KUKA KRL program: EPS_2_251806_MH47A_A_20260212042244.src

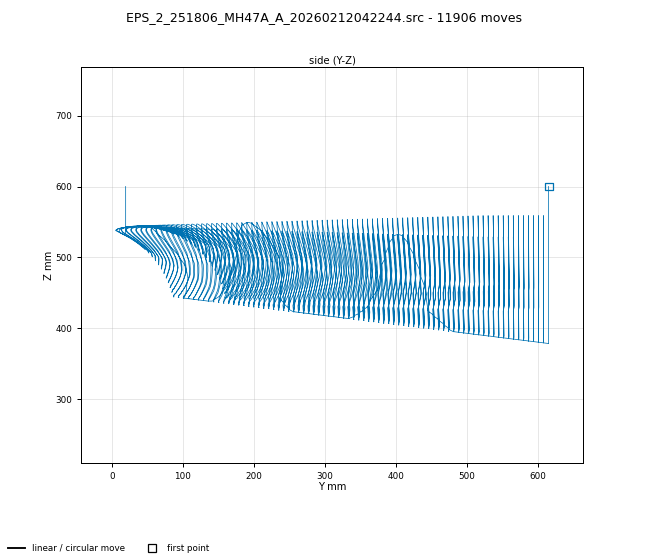
[picture p0: tool path of EPS_2_251806_MH47A_A_20260212042244.src, 11906 of 11908 moves have a stored position in this frame; points joined in program order, loops and branches not executed]
&ACCESS RVP
&REL 4
&COMMENT QRS 19112012
&PARAM EDITMASK = *
DEF PART()
EXT BAS (BAS_COMMAND :IN,REAL :IN )
INT I
BAS (#INITMOV,0 )

;KUKA QRS Post kuka4.cps  Date:22-06-2017 !

File_ID=3019

QRS_PRE_INIT()

;Init var - Until changes are made in qrs_pre_init
Outlet_Square_prg=0
Inlet_1_Square_prg=0
Inlet_2_Square_prg=0
Inlet_3_Square_prg=0
Inlet_4_Square_prg=0
Inlet_5_Square_prg=0

Outlet_1={X 0.000, Y 520.860, Z 458.500, B 0.000, E1 0.000 }
Inlet_1={X 0.000, Y 523.030, Z 428.500, B 0.000, E1 194.000 }
Outlet_1_type=201
Inlet_1_type=201
;QRS#1=Sidecore dimensions
;QRS#2=200-8" PVC SDR 35
;QRS#3=200-8" PVC SDR 35
;QRS#4=
;QRS#5=
;QRS#6=
;QRS#7=
;QRS#8=
;QRS#9=12-08 PSX
;QRS#10=12-08 PSX
;QRS#11=
;QRS#12=
;QRS#13=
;QRS#14=
;QRS#15=
;QRS#16=1220x127x838 2,75'
;QRS#17=EPS Height
;QRS#18=559
;QRS#19=*
;QRS#20= UPDATED VERSION 22-06-2017
;QRS#21=*
Outlet_Square=0100
Inlet_1_Square=0100
Inlet_2_Square=0
Inlet_3_Square=0
Inlet_4_Square=0
Inlet_5_Square=0
Mill_Square=1
Outlet_Square_Prg=204
Inlet_1_Square_prg=204

QRS_INIT()

$ADVANCE=5

; T1
PTP {E1 173.598,E2 173.598}
PTP {X 0,Y 615.497,A -85,B 0,C 180,E1 173.598,E2 173.598,E3 0,E4 0,E5 0,E6 0}
QRS_SPEED_INIT()
LIN {X 0,Y 615.497,Z 600,A -85,B 0,C 180,E1 173.598,E2 173.598,E3 0,E4 0,E5 0,E6 0} C_VEL
LIN {X 0,Y 615.497,Z 388.866,A -85,B 0,C 180,E1 173.598,E2 173.598} C_VEL
LIN {X 0,Y 615.497,Z 380.69,A -85,B 0,C 180,E1 173.598,E2 173.598} C_VEL
LIN {X 0,Y 615.486,Z 378.69,A -85,B 0,C 180,E1 173.412,E2 173.412} C_VEL
LIN {X 0,Y 615.496,Z 378.692,A -85,B 0,C 180,E1 170.801,E2 170.801} C_VEL
LIN {X 0,Y 615.477,Z 378.685,A -85,B 0,C 180,E1 168.139,E2 168.139} C_VEL
LIN {X 0,Y 615.488,Z 378.696,A -85,B 0,C 180,E1 165.451,E2 165.451} C_VEL
LIN {X 0,Y 615.493,Z 378.685,A -85,B 0,C 180,E1 162.73,E2 162.73} C_VEL
LIN {X 0,Y 615.49,Z 378.687,A -85,B 0,C 180,E1 159.967,E2 159.967} C_VEL
LIN {X 0,Y 615.491,Z 378.69,A -85,B 0,C 180,E1 157.156,E2 157.156} C_VEL
LIN {X 0,Y 615.475,Z 378.687,A -85,B 0,C 180,E1 154.431,E2 154.431} C_VEL
LIN {X 0,Y 615.483,Z 378.692,A -85,B 0,C 180,E1 152.085,E2 152.085} C_VEL
LIN {X 0,Y 615.49,Z 378.7,A -85,B 0,C 180,E1 149.84,E2 149.84} C_VEL
LIN {X 0,Y 615.485,Z 378.693,A -85,B 0,C 180,E1 147.542,E2 147.542} C_VEL
LIN {X 0,Y 615.492,Z 378.683,A -85,B 0,C 180,E1 145.185,E2 145.185} C_VEL
LIN {X 0,Y 615.479,Z 378.686,A -85,B 0,C 180,E1 142.757,E2 142.757} C_VEL
LIN {X 0,Y 615.486,Z 378.696,A -85,B 0,C 180,E1 139.91,E2 139.91} C_VEL
LIN {X 0,Y 615.483,Z 378.686,A -85,B 0,C 180,E1 136.952,E2 136.952} C_VEL
LIN {X 0,Y 615.482,Z 378.693,A -85,B 0,C 180,E1 133.997,E2 133.997} C_VEL
LIN {X 0,Y 615.488,Z 378.683,A -85,B 0,C 180,E1 131.473,E2 131.473} C_VEL
LIN {X 0,Y 615.484,Z 378.691,A -85,B 0,C 180,E1 128.903,E2 128.903} C_VEL
LIN {X 0,Y 615.49,Z 378.696,A -85,B 0,C 180,E1 126.424,E2 126.424} C_VEL
LIN {X 0,Y 615.492,Z 378.683,A -85,B 0,C 180,E1 123.535,E2 123.535} C_VEL
LIN {X 0,Y 615.493,Z 378.697,A -85,B 0,C 180,E1 120.919,E2 120.919} C_VEL
LIN {X 0,Y 615.491,Z 378.689,A -85,B 0,C 180,E1 118.451,E2 118.451} C_VEL
LIN {X 0,Y 615.498,Z 378.684,A -85,B 0,C 180,E1 115.571,E2 115.571} C_VEL
LIN {X 0,Y 615.494,Z 378.694,A -85,B 0,C 180,E1 112.844,E2 112.844} C_VEL
LIN {X 0,Y 615.494,Z 378.691,A -85,B 0,C 180,E1 111.431,E2 111.431} C_VEL
LIN {X 0,Y 615.49,Z 382.133,A -85,B 0,C 180,E1 109.337,E2 109.337} C_VEL
LIN {X 0,Y 615.489,Z 386.996,A -85,B 0,C 180,E1 106.586,E2 106.586} C_VEL
LIN {X 0,Y 615.492,Z 391.972,A -85,B 0,C 180,E1 103.874,E2 103.874} C_VEL
LIN {X 0,Y 615.494,Z 397.582,A -85,B 0,C 180,E1 100.891,E2 100.891} C_VEL
LIN {X 0,Y 615.48,Z 402.111,A -85,B 0,C 180,E1 98.536,E2 98.536} C_VEL
LIN {X 0,Y 615.498,Z 407.278,A -85,B 0,C 180,E1 95.898,E2 95.898} C_VEL
LIN {X 0,Y 615.485,Z 412.5,A -85,B 0,C 180,E1 93.273,E2 93.273} C_VEL
LIN {X 0,Y 615.48,Z 417.779,A -85,B 0,C 180,E1 90.654,E2 90.654} C_VEL
LIN {X 0,Y 615.499,Z 423.128,A -85,B 0,C 180,E1 88.037,E2 88.037} C_VEL
LIN {X 0,Y 615.492,Z 424.091,A -85,B 0,C 180,E1 87.566,E2 87.566} C_VEL
LIN {X 0,Y 615.493,Z 439.332,A -85,B 0,C 180,E1 87.218,E2 87.218} C_VEL
LIN {X 0,Y 615.483,Z 451.508,A -85,B 0,C 180,E1 86.809,E2 86.809} C_VEL
LIN {X 0,Y 615.483,Z 462.446,A -85,B 0,C 180,E1 86.317,E2 86.317} C_VEL
LIN {X 0,Y 615.492,Z 473.835,A -85,B 0,C 180,E1 85.662,E2 85.662} C_VEL
LIN {X 0,Y 615.498,Z 484.113,A -85,B 0,C 180,E1 84.923,E2 84.923} C_VEL
LIN {X 0,Y 615.5,Z 493.432,A -85,B 0,C 180,E1 84.102,E2 84.102} C_VEL
LIN {X 0,Y 615.496,Z 502.546,A -85,B 0,C 180,E1 83.1,E2 83.1} C_VEL
LIN {X 0,Y 615.497,Z 509.707,A -85,B 0,C 180,E1 82.125,E2 82.125} C_VEL
LIN {X 0,Y 615.496,Z 515.553,A -85,B 0,C 180,E1 81.133,E2 81.133} C_VEL
LIN {X 0,Y 615.499,Z 520.165,A -85,B 0,C 180,E1 80.138,E2 80.138} C_VEL
LIN {X 0,Y 615.495,Z 523.781,A -85,B 0,C 180,E1 79.109,E2 79.109} C_VEL
LIN {X 0,Y 615.496,Z 526.184,A -85,B 0,C 180,E1 78.139,E2 78.139} C_VEL
LIN {X 0,Y 615.494,Z 527.337,A -85,B 0,C 180,E1 77.47,E2 77.47} C_VEL
LIN {X 0,Y 615.496,Z 528.353,A -85,B 0,C 180,E1 76.126,E2 76.126} C_VEL
LIN {X 0,Y 615.497,Z 528.272,A -85,B 0,C 180,E1 75.451,E2 75.451} C_VEL
LIN {X 0,Y 615.494,Z 527.732,A -85,B 0,C 180,E1 74.774,E2 74.774} C_VEL
LIN {X 0,Y 615.493,Z 525.744,A -85,B 0,C 180,E1 73.567,E2 73.567} C_VEL
LIN {X 0,Y 615.498,Z 522.455,A -85,B 0,C 180,E1 72.387,E2 72.387} C_VEL
LIN {X 0,Y 615.497,Z 518.373,A -85,B 0,C 180,E1 71.355,E2 71.355} C_VEL
LIN {X 0,Y 615.497,Z 511.943,A -85,B 0,C 180,E1 70.142,E2 70.142} C_VEL
LIN {X 0,Y 615.498,Z 504.805,A -85,B 0,C 180,E1 69.095,E2 69.095} C_VEL
LIN {X 0,Y 615.499,Z 497.407,A -85,B 0,C 180,E1 68.217,E2 68.217} C_VEL
LIN {X 0,Y 615.5,Z 489.091,A -85,B 0,C 180,E1 67.404,E2 67.404} C_VEL
LIN {X 0,Y 615.5,Z 479.313,A -85,B 0,C 180,E1 66.623,E2 66.623} C_VEL
LIN {X 0,Y 615.477,Z 468.588,A -85,B 0,C 180,E1 65.927,E2 65.927} C_VEL
LIN {X 0,Y 615.488,Z 456.806,A -85,B 0,C 180,E1 65.324,E2 65.324} C_VEL
LIN {X 0,Y 615.478,Z 444.92,A -85,B 0,C 180,E1 64.863,E2 64.863} C_VEL
LIN {X 0,Y 615.495,Z 431.787,A -85,B 0,C 180,E1 64.502,E2 64.502} C_VEL
LIN {X 0,Y 615.491,Z 424.082,A -85,B 0,C 180,E1 64.339,E2 64.339} C_VEL
LIN {X 0,Y 615.491,Z 418.375,A -85,B 0,C 180,E1 61.549,E2 61.549} C_VEL
LIN {X 0,Y 615.478,Z 413.056,A -85,B 0,C 180,E1 58.915,E2 58.915} C_VEL
LIN {X 0,Y 615.492,Z 408.176,A -85,B 0,C 180,E1 56.465,E2 56.465} C_VEL
LIN {X 0,Y 615.485,Z 402.503,A -85,B 0,C 180,E1 53.576,E2 53.576} C_VEL
LIN {X 0,Y 615.488,Z 397.43,A -85,B 0,C 180,E1 50.938,E2 50.938} C_VEL
LIN {X 0,Y 615.488,Z 392.894,A -85,B 0,C 180,E1 48.527,E2 48.527} C_VEL
LIN {X 0,Y 615.491,Z 387.954,A -85,B 0,C 180,E1 45.852,E2 45.852} C_VEL
LIN {X 0,Y 615.489,Z 382.969,A -85,B 0,C 180,E1 43.049,E2 43.049} C_VEL
LIN {X 0,Y 615.481,Z 378.717,A -85,B 0,C 180,E1 40.607,E2 40.607} C_VEL
LIN {X 0,Y 615.483,Z 378.698,A -85,B 0,C 180,E1 38.013,E2 38.013} C_VEL
LIN {X 0,Y 615.48,Z 378.693,A -85,B 0,C 180,E1 35.616,E2 35.616} C_VEL
LIN {X 0,Y 615.494,Z 378.699,A -85,B 0,C 180,E1 33.236,E2 33.236} C_VEL
LIN {X 0,Y 615.49,Z 378.691,A -85,B 0,C 180,E1 30.919,E2 30.919} C_VEL
LIN {X 0,Y 615.483,Z 378.695,A -85,B 0,C 180,E1 28.451,E2 28.451} C_VEL
LIN {X 0,Y 615.493,Z 378.698,A -85,B 0,C 180,E1 25.715,E2 25.715} C_VEL
LIN {X 0,Y 615.488,Z 378.702,A -85,B 0,C 180,E1 22.844,E2 22.844} C_VEL
LIN {X 0,Y 615.497,Z 378.696,A -85,B 0,C 180,E1 20.032,E2 20.032} C_VEL
LIN {X 0,Y 615.492,Z 378.693,A -85,B 0,C 180,E1 17.27,E2 17.27} C_VEL
LIN {X 0,Y 615.481,Z 378.693,A -85,B 0,C 180,E1 14.549,E2 14.549} C_VEL
LIN {X 0,Y 615.477,Z 378.694,A -85,B 0,C 180,E1 11.861,E2 11.861} C_VEL
LIN {X 0,Y 615.489,Z 378.697,A -85,B 0,C 180,E1 9.199,E2 9.199} C_VEL
LIN {X 0,Y 615.489,Z 378.699,A -85,B 0,C 180,E1 6.557,E2 6.557} C_VEL
LIN {X 0,Y 615.477,Z 378.695,A -85,B 0,C 180,E1 3.928,E2 3.928} C_VEL
LIN {X 0,Y 615.487,Z 378.691,A -85,B 0,C 180,E1 1.308,E2 1.308} C_VEL
LIN {X 0,Y 615.491,Z 378.695,A -85,B 0,C 180,E1 -1.309,E2 -1.309} C_VEL
LIN {X 0,Y 615.488,Z 378.7,A -85,B 0,C 180,E1 -3.929,E2 -3.929} C_VEL
LIN {X 0,Y 615.492,Z 378.692,A -85,B 0,C 180,E1 -6.591,E2 -6.591} C_VEL
LIN {X 0,Y 615.489,Z 378.691,A -85,B 0,C 180,E1 -9.199,E2 -9.199} C_VEL
LIN {X 0,Y 615.486,Z 378.695,A -85,B 0,C 180,E1 -11.861,E2 -11.861} C_VEL
LIN {X 0,Y 615.492,Z 378.7,A -85,B 0,C 180,E1 -14.549,E2 -14.549} C_VEL
LIN {X 0,Y 615.492,Z 378.696,A -85,B 0,C 180,E1 -17.271,E2 -17.271} C_VEL
LIN {X 0,Y 615.49,Z 378.693,A -85,B 0,C 180,E1 -20.033,E2 -20.033} C_VEL
LIN {X 0,Y 615.481,Z 378.693,A -85,B 0,C 180,E1 -22.845,E2 -22.845} C_VEL
LIN {X 0,Y 615.475,Z 378.694,A -85,B 0,C 180,E1 -25.568,E2 -25.568} C_VEL
LIN {X 0,Y 615.483,Z 378.703,A -85,B 0,C 180,E1 -27.915,E2 -27.915} C_VEL
LIN {X 0,Y 615.489,Z 378.691,A -85,B 0,C 180,E1 -30.16,E2 -30.16} C_VEL
LIN {X 0,Y 615.494,Z 378.7,A -85,B 0,C 180,E1 -32.457,E2 -32.457} C_VEL
LIN {X 0,Y 615.49,Z 378.691,A -85,B 0,C 180,E1 -34.815,E2 -34.815} C_VEL
LIN {X 0,Y 615.48,Z 378.696,A -85,B 0,C 180,E1 -37.243,E2 -37.243} C_VEL
LIN {X 0,Y 615.483,Z 378.699,A -85,B 0,C 180,E1 -40.09,E2 -40.09} C_VEL
LIN {X 0,Y 615.477,Z 378.694,A -85,B 0,C 180,E1 -42.354,E2 -42.354} C_VEL
LIN {X 0,Y 615.479,Z 378.693,A -85,B 0,C 180,E1 -45.07,E2 -45.07} C_VEL
LIN {X 0,Y 615.485,Z 378.693,A -85,B 0,C 180,E1 -47.92,E2 -47.92} C_VEL
LIN {X 0,Y 615.495,Z 378.698,A -85,B 0,C 180,E1 -50.251,E2 -50.251} C_VEL
LIN {X 0,Y 615.486,Z 378.696,A -85,B 0,C 180,E1 -53.064,E2 -53.064} C_VEL
LIN {X 0,Y 615.49,Z 378.81,A -85,B 0,C 180,E1 -54.586,E2 -54.586} C_VEL
LIN {X 0,Y 615.495,Z 387.116,A -85,B 0,C 180,E1 -57.544,E2 -57.544} C_VEL
LIN {X 0,Y 615.479,Z 394.86,A -85,B 0,C 180,E1 -60.207,E2 -60.207} C_VEL
LIN {X 0,Y 615.478,Z 403.061,A -85,B 0,C 180,E1 -62.957,E2 -62.957} C_VEL
LIN {X 0,Y 615.495,Z 411.524,A -85,B 0,C 180,E1 -65.729,E2 -65.729} C_VEL
LIN {X 0,Y 615.485,Z 420.391,A -85,B 0,C 180,E1 -68.568,E2 -68.568} C_VEL
LIN {X 0,Y 615.488,Z 429.381,A -85,B 0,C 180,E1 -71.396,E2 -71.396} C_VEL
LIN {X 0,Y 615.484,Z 438.109,A -85,B 0,C 180,E1 -74.095,E2 -74.095} C_VEL
LIN {X 0,Y 615.495,Z 446.951,A -85,B 0,C 180,E1 -76.799,E2 -76.799} C_VEL
LIN {X 0,Y 615.491,Z 452.138,A -85,B 0,C 180,E1 -78.369,E2 -78.369} C_VEL
LIN {X 0,Y 615.499,Z 465.825,A -85,B 0,C 180,E1 -78.64,E2 -78.64} C_VEL
LIN {X 0,Y 615.489,Z 478.536,A -85,B 0,C 180,E1 -79.036,E2 -79.036} C_VEL
LIN {X 0,Y 615.479,Z 490.769,A -85,B 0,C 180,E1 -79.556,E2 -79.556} C_VEL
LIN {X 0,Y 615.498,Z 501.388,A -85,B 0,C 180,E1 -80.138,E2 -80.138} C_VEL
LIN {X 0,Y 615.498,Z 512.232,A -85,B 0,C 180,E1 -80.884,E2 -80.884} C_VEL
LIN {X 0,Y 615.497,Z 522.812,A -85,B 0,C 180,E1 -81.794,E2 -81.794} C_VEL
LIN {X 0,Y 615.498,Z 530.606,A -85,B 0,C 180,E1 -82.62,E2 -82.62} C_VEL
LIN {X 0,Y 615.496,Z 538.203,A -85,B 0,C 180,E1 -83.608,E2 -83.608} C_VEL
LIN {X 0,Y 615.498,Z 545.204,A -85,B 0,C 180,E1 -84.759,E2 -84.759} C_VEL
LIN {X 0,Y 615.493,Z 549.851,A -85,B 0,C 180,E1 -85.744,E2 -85.744} C_VEL
LIN {X 0,Y 615.495,Z 553.398,A -85,B 0,C 180,E1 -86.727,E2 -86.727} C_VEL
LIN {X 0,Y 615.497,Z 555.233,A -85,B 0,C 180,E1 -87.382,E2 -87.382} C_VEL
LIN {X 0,Y 615.499,Z 556.607,A -85,B 0,C 180,E1 -88.037,E2 -88.037} C_VEL
LIN {X 0,Y 615.496,Z 558.173,A -85,B 0,C 180,E1 -89.346,E2 -89.346} C_VEL
LIN {X 0,Y 615.494,Z 558.389,A -85,B 0,C 180,E1 -90,E2 -90} C_VEL
LIN {X 0,Y 615.496,Z 557.58,A -85,B 0,C 180,E1 -91.308,E2 -91.308} C_VEL
LIN {X 0,Y 615.499,Z 556.608,A -85,B 0,C 180,E1 -91.963,E2 -91.963} C_VEL
LIN {X 0,Y 615.497,Z 555.233,A -85,B 0,C 180,E1 -92.618,E2 -92.618} C_VEL
LIN {X 0,Y 615.496,Z 552.35,A -85,B 0,C 180,E1 -93.6,E2 -93.6} C_VEL
LIN {X 0,Y 615.498,Z 548.442,A -85,B 0,C 180,E1 -94.584,E2 -94.584} C_VEL
LIN {X 0,Y 615.499,Z 543.406,A -85,B 0,C 180,E1 -95.569,E2 -95.569} C_VEL
LIN {X 0,Y 615.497,Z 536.87,A -85,B 0,C 180,E1 -96.583,E2 -96.583} C_VEL
LIN {X 0,Y 615.497,Z 529.136,A -85,B 0,C 180,E1 -97.545,E2 -97.545} C_VEL
LIN {X 0,Y 615.498,Z 521.048,A -85,B 0,C 180,E1 -98.371,E2 -98.371} C_VEL
LIN {X 0,Y 615.499,Z 511.172,A -85,B 0,C 180,E1 -99.198,E2 -99.198} C_VEL
LIN {X 0,Y 615.491,Z 499.986,A -85,B 0,C 180,E1 -99.945,E2 -99.945} C_VEL
LIN {X 0,Y 615.481,Z 489.031,A -85,B 0,C 180,E1 -100.527,E2 -100.527} C_VEL
LIN {X 0,Y 615.489,Z 476.475,A -85,B 0,C 180,E1 -101.04,E2 -101.04} C_VEL
LIN {X 0,Y 615.498,Z 464.079,A -85,B 0,C 180,E1 -101.401,E2 -101.401} C_VEL
LIN {X 0,Y 615.491,Z 452.139,A -85,B 0,C 180,E1 -101.631,E2 -101.631} C_VEL
LIN {X 0,Y 615.476,Z 443.545,A -85,B 0,C 180,E1 -104.24,E2 -104.24} C_VEL
LIN {X 0,Y 615.483,Z 434.785,A -85,B 0,C 180,E1 -106.928,E2 -106.928} C_VEL
LIN {X 0,Y 615.485,Z 425.93,A -85,B 0,C 180,E1 -109.684,E2 -109.684} C_VEL
LIN {X 0,Y 615.491,Z 417.513,A -85,B 0,C 180,E1 -112.346,E2 -112.346} C_VEL
LIN {X 0,Y 615.478,Z 409.311,A -85,B 0,C 180,E1 -114.991,E2 -114.991} C_VEL
LIN {X 0,Y 615.494,Z 401.544,A -85,B 0,C 180,E1 -117.544,E2 -117.544} C_VEL
LIN {X 0,Y 615.497,Z 392.671,A -85,B 0,C 180,E1 -120.538,E2 -120.538} C_VEL
LIN {X 0,Y 615.491,Z 384.892,A -85,B 0,C 180,E1 -123.235,E2 -123.235} C_VEL
LIN {X 0,Y 615.49,Z 378.691,A -85,B 0,C 180,E1 -125.514,E2 -125.514} C_VEL
LIN {X 0,Y 615.481,Z 378.685,A -85,B 0,C 180,E1 -128.068,E2 -128.068} C_VEL
LIN {X 0,Y 615.491,Z 378.69,A -85,B 0,C 180,E1 -130.605,E2 -130.605} C_VEL
LIN {X 0,Y 615.496,Z 378.689,A -85,B 0,C 180,E1 -133.243,E2 -133.243} C_VEL
LIN {X 0,Y 615.484,Z 378.685,A -85,B 0,C 180,E1 -136.002,E2 -136.002} C_VEL
LIN {X 0,Y 615.492,Z 378.694,A -85,B 0,C 180,E1 -138.903,E2 -138.903} C_VEL
LIN {X 0,Y 615.49,Z 378.688,A -85,B 0,C 180,E1 -141.096,E2 -141.096} C_VEL
LIN {X 0,Y 615.478,Z 378.685,A -85,B 0,C 180,E1 -143.574,E2 -143.574} C_VEL
LIN {X 0,Y 615.492,Z 378.7,A -85,B 0,C 180,E1 -146.463,E2 -146.463} C_VEL
LIN {X 0,Y 615.487,Z 378.685,A -85,B 0,C 180,E1 -149.08,E2 -149.08} C_VEL
LIN {X 0,Y 615.478,Z 378.687,A -85,B 0,C 180,E1 -151.549,E2 -151.549} C_VEL
LIN {X 0,Y 615.478,Z 378.7,A -85,B 0,C 180,E1 -154.284,E2 -154.284} C_VEL
LIN {X 0,Y 615.475,Z 378.694,A -85,B 0,C 180,E1 -156.443,E2 -156.443} C_VEL
LIN {X 0,Y 615.479,Z 378.689,A -85,B 0,C 180,E1 -158.568,E2 -158.568} C_VEL
LIN {X 0,Y 615.477,Z 378.69,A -85,B 0,C 180,E1 -161.394,E2 -161.394} C_VEL
LIN {X 0,Y 615.476,Z 378.696,A -85,B 0,C 180,E1 -164.094,E2 -164.094} C_VEL
LIN {X 0,Y 615.494,Z 378.682,A -85,B 0,C 180,E1 -166.799,E2 -166.799} C_VEL
LIN {X 0,Y 615.486,Z 378.698,A -85,B 0,C 180,E1 -169.473,E2 -169.473} C_VEL
LIN {X 0,Y 615.478,Z 378.689,A -85,B 0,C 180,E1 -172.124,E2 -172.124} C_VEL
LIN {X 0,Y 615.487,Z 378.685,A -85,B 0,C 180,E1 -174.759,E2 -174.759} C_VEL
LIN {X 0,Y 615.495,Z 378.7,A -85,B 0,C 180,E1 -177.382,E2 -177.382} C_VEL
LIN {X 0,Y 615.478,Z 378.687,A -85,B 0,C 180,E1 -180,E2 -180} C_VEL
LIN {X 0,Y 615.488,Z 378.687,A -85,B 0,C 180,E1 -182.618,E2 -182.618} C_VEL
LIN {X 0,Y 615.495,Z 378.696,A -85,B 0,C 180,E1 -185.241,E2 -185.241} C_VEL
LIN {X 0,Y 615.486,Z 378.69,A -85,B 0,C 180,E1 -186.588,E2 -186.588} C_VEL
LIN {X 0,Y 614.813,Z 378.842,A -85,B 0,C 180,E1 -187.134,E2 -187.134} C_VEL
LIN {X 0,Y 611.985,Z 379.248,A -85,B 0,C 180,E1 -188.02,E2 -188.02} C_VEL
LIN {X 0,Y 609.593,Z 379.559,A -85,B 0,C 180,E1 -188.732,E2 -188.732} C_VEL
LIN {X 0,Y 608.554,Z 379.68,A -85,B 0,C 180,E1 -189.282,E2 -189.282} C_VEL
LIN {X 0,Y 608.461,Z 379.689,A -85,B 0,C 180,E1 -189.468,E2 -189.468} C_VEL
LIN {X 0,Y 608.454,Z 379.688,A -85,B 0,C 180,E1 -192,E2 -192} C_VEL
LIN {X 0,Y 608.475,Z 379.695,A -85,B 0,C 180,E1 -194.72,E2 -194.72} C_VEL
LIN {X 0,Y 608.454,Z 379.688,A -85,B 0,C 180,E1 -197.476,E2 -197.476} C_VEL
LIN {X 0,Y 608.465,Z 379.692,A -85,B 0,C 180,E1 -200.274,E2 -200.274} C_VEL
LIN {X 0,Y 608.448,Z 379.69,A -85,B 0,C 180,E1 -203.124,E2 -203.124} C_VEL
LIN {X 0,Y 608.462,Z 379.688,A -85,B 0,C 180,E1 -205.722,E2 -205.722} C_VEL
LIN {X 0,Y 608.454,Z 379.698,A -85,B 0,C 180,E1 -208.266,E2 -208.266} C_VEL
LIN {X 0,Y 608.473,Z 379.69,A -85,B 0,C 180,E1 -210.545,E2 -210.545} C_VEL
LIN {X 0,Y 608.454,Z 379.688,A -85,B 0,C 180,E1 -212.88,E2 -212.88} C_VEL
LIN {X 0,Y 608.442,Z 379.69,A -85,B 0,C 180,E1 -215.278,E2 -215.278} C_VEL
LIN {X 0,Y 608.467,Z 379.693,A -85,B 0,C 180,E1 -217.746,E2 -217.746} C_VEL
LIN {X 0,Y 608.449,Z 379.691,A -85,B 0,C 180,E1 -220.33,E2 -220.33} C_VEL
LIN {X 0,Y 608.449,Z 379.689,A -85,B 0,C 180,E1 -222.96,E2 -222.96} C_VEL
LIN {X 0,Y 608.458,Z 379.697,A -85,B 0,C 180,E1 -225.736,E2 -225.736} C_VEL
LIN {X 0,Y 608.463,Z 379.686,A -85,B 0,C 180,E1 -228.658,E2 -228.658} C_VEL
LIN {X 0,Y 608.466,Z 379.695,A -85,B 0,C 180,E1 -231.413,E2 -231.413} C_VEL
LIN {X 0,Y 608.473,Z 379.687,A -85,B 0,C 180,E1 -233.951,E2 -233.951} C_VEL
LIN {X 0,Y 608.465,Z 379.686,A -85,B 0,C 180,E1 -236.33,E2 -236.33} C_VEL
LIN {X 0,Y 608.477,Z 379.687,A -85,B 0,C 180,E1 -238.728,E2 -238.728} C_VEL
LIN {X 0,Y 608.476,Z 379.691,A -85,B 0,C 180,E1 -241.38,E2 -241.38} C_VEL
LIN {X 0,Y 608.446,Z 379.689,A -85,B 0,C 180,E1 -243.965,E2 -243.965} C_VEL
LIN {X 0,Y 608.463,Z 379.687,A -85,B 0,C 180,E1 -246.156,E2 -246.156} C_VEL
LIN {X 0,Y 608.47,Z 379.687,A -85,B 0,C 180,E1 -248.309,E2 -248.309} C_VEL
LIN {X 0,Y 608.467,Z 380.749,A -85,B 0,C 180,E1 -249.322,E2 -249.322} C_VEL
LIN {X 0,Y 608.454,Z 385.12,A -85,B 0,C 180,E1 -251.829,E2 -251.829} C_VEL
LIN {X 0,Y 608.447,Z 390.041,A -85,B 0,C 180,E1 -254.594,E2 -254.594} C_VEL
LIN {X 0,Y 608.449,Z 395.071,A -85,B 0,C 180,E1 -257.323,E2 -257.323} C_VEL
LIN {X 0,Y 608.465,Z 400.167,A -85,B 0,C 180,E1 -260.023,E2 -260.023} C_VEL
LIN {X 0,Y 608.451,Z 405.329,A -85,B 0,C 180,E1 -262.701,E2 -262.701} C_VEL
LIN {X 0,Y 608.448,Z 410.555,A -85,B 0,C 180,E1 -265.363,E2 -265.363} C_VEL
LIN {X 0,Y 608.443,Z 415.843,A -85,B 0,C 180,E1 -268.014,E2 -268.014} C_VEL
LIN {X 0,Y 608.43,Z 421.193,A -85,B 0,C 180,E1 -270.662,E2 -270.662} C_VEL
LIN {X 0,Y 608.427,Z 424.526,A -85,B 0,C 180,E1 -272.296,E2 -272.296} C_VEL
LIN {X 0,Y 608.527,Z 440.823,A -85,B 0,C 180,E1 -272.689,E2 -272.689} C_VEL
LIN {X 0,Y 608.506,Z 453.546,A -85,B 0,C 180,E1 -273.145,E2 -273.145} C_VEL
LIN {X 0,Y 608.508,Z 465.634,A -85,B 0,C 180,E1 -273.725,E2 -273.725} C_VEL
LIN {X 0,Y 608.481,Z 476.518,A -85,B 0,C 180,E1 -274.389,E2 -274.389} C_VEL
LIN {X 0,Y 608.483,Z 486.366,A -85,B 0,C 180,E1 -275.136,E2 -275.136} C_VEL
LIN {X 0,Y 608.456,Z 495.335,A -85,B 0,C 180,E1 -275.967,E2 -275.967} C_VEL
LIN {X 0,Y 608.463,Z 504.126,A -85,B 0,C 180,E1 -276.966,E2 -276.966} C_VEL
LIN {X 0,Y 608.439,Z 511.195,A -85,B 0,C 180,E1 -277.967,E2 -277.967} C_VEL
LIN {X 0,Y 608.447,Z 516.858,A -85,B 0,C 180,E1 -278.971,E2 -278.971} C_VEL
LIN {X 0,Y 608.437,Z 521.328,A -85,B 0,C 180,E1 -279.978,E2 -279.978} C_VEL
LIN {X 0,Y 608.452,Z 524.61,A -85,B 0,C 180,E1 -280.947,E2 -280.947} C_VEL
LIN {X 0,Y 608.44,Z 527.103,A -85,B 0,C 180,E1 -282,E2 -282} C_VEL
LIN {X 0,Y 608.44,Z 528.765,A -85,B 0,C 180,E1 -283.357,E2 -283.357} C_VEL
LIN {X 0,Y 608.424,Z 529,A -85,B 0,C 180,E1 -284.038,E2 -284.038} C_VEL
LIN {X 0,Y 608.418,Z 528.773,A -85,B 0,C 180,E1 -284.722,E2 -284.722} C_VEL
LIN {X 0,Y 608.417,Z 528.139,A -85,B 0,C 180,E1 -285.407,E2 -285.407} C_VEL
LIN {X 0,Y 608.422,Z 526.211,A -85,B 0,C 180,E1 -286.514,E2 -286.514} C_VEL
LIN {X 0,Y 608.428,Z 522.402,A -85,B 0,C 180,E1 -287.824,E2 -287.824} C_VEL
LIN {X 0,Y 608.457,Z 518.072,A -85,B 0,C 180,E1 -288.869,E2 -288.869} C_VEL
LIN {X 0,Y 608.437,Z 512.411,A -85,B 0,C 180,E1 -289.922,E2 -289.922} C_VEL
LIN {X 0,Y 608.472,Z 505.222,A -85,B 0,C 180,E1 -290.981,E2 -290.981} C_VEL
LIN {X 0,Y 608.455,Z 497.769,A -85,B 0,C 180,E1 -291.87,E2 -291.87} C_VEL
LIN {X 0,Y 608.471,Z 487.852,A -85,B 0,C 180,E1 -292.826,E2 -292.826} C_VEL
LIN {X 0,Y 608.496,Z 477.085,A -85,B 0,C 180,E1 -293.663,E2 -293.663} C_VEL
LIN {X 0,Y 608.501,Z 465.339,A -85,B 0,C 180,E1 -294.381,E2 -294.381} C_VEL
LIN {X 0,Y 608.5,Z 452.765,A -85,B 0,C 180,E1 -294.979,E2 -294.979} C_VEL
LIN {X 0,Y 608.518,Z 439.923,A -85,B 0,C 180,E1 -295.426,E2 -295.426} C_VEL
LIN {X 0,Y 608.567,Z 426.488,A -85,B 0,C 180,E1 -295.739,E2 -295.739} C_VEL
LIN {X 0,Y 608.424,Z 424.525,A -85,B 0,C 180,E1 -295.794,E2 -295.794} C_VEL
LIN {X 0,Y 608.424,Z 418.794,A -85,B 0,C 180,E1 -298.611,E2 -298.611} C_VEL
LIN {X 0,Y 608.414,Z 413.356,A -85,B 0,C 180,E1 -301.319,E2 -301.319} C_VEL
LIN {X 0,Y 608.425,Z 408.581,A -85,B 0,C 180,E1 -303.728,E2 -303.728} C_VEL
LIN {X 0,Y 608.444,Z 403.966,A -85,B 0,C 180,E1 -306.092,E2 -306.092} C_VEL
LIN {X 0,Y 608.432,Z 399.173,A -85,B 0,C 180,E1 -308.59,E2 -308.59} C_VEL
LIN {X 0,Y 608.435,Z 394.007,A -85,B 0,C 180,E1 -311.339,E2 -311.339} C_VEL
LIN {X 0,Y 608.459,Z 388.648,A -85,B 0,C 180,E1 -314.264,E2 -314.264} C_VEL
LIN {X 0,Y 608.451,Z 383.748,A -85,B 0,C 180,E1 -317.04,E2 -317.04} C_VEL
LIN {X 0,Y 608.444,Z 380.67,A -85,B 0,C 180,E1 -318.823,E2 -318.823} C_VEL
LIN {X 0,Y 608.446,Z 379.694,A -85,B 0,C 180,E1 -319.696,E2 -319.696} C_VEL
LIN {X 0,Y 608.466,Z 379.696,A -85,B 0,C 180,E1 -322.254,E2 -322.254} C_VEL
LIN {X 0,Y 608.486,Z 379.693,A -85,B 0,C 180,E1 -325.088,E2 -325.088} C_VEL
LIN {X 0,Y 608.462,Z 379.694,A -85,B 0,C 180,E1 -327.905,E2 -327.905} C_VEL
LIN {X 0,Y 608.47,Z 379.69,A -85,B 0,C 180,E1 -330.221,E2 -330.221} C_VEL
LIN {X 0,Y 608.485,Z 379.692,A -85,B 0,C 180,E1 -332.79,E2 -332.79} C_VEL
LIN {X 0,Y 608.46,Z 379.694,A -85,B 0,C 180,E1 -335.429,E2 -335.429} C_VEL
LIN {X 0,Y 608.473,Z 379.691,A -85,B 0,C 180,E1 -338.309,E2 -338.309} C_VEL
LIN {X 0,Y 608.468,Z 379.692,A -85,B 0,C 180,E1 -341.282,E2 -341.282} C_VEL
LIN {X 0,Y 608.457,Z 379.691,A -85,B 0,C 180,E1 -343.906,E2 -343.906} C_VEL
LIN {X 0,Y 608.472,Z 379.69,A -85,B 0,C 180,E1 -346.644,E2 -346.644} C_VEL
LIN {X 0,Y 608.465,Z 379.693,A -85,B 0,C 180,E1 -349.35,E2 -349.35} C_VEL
LIN {X 0,Y 608.477,Z 379.695,A -85,B 0,C 180,E1 -352.033,E2 -352.033} C_VEL
LIN {X 0,Y 608.472,Z 379.691,A -85,B 0,C 180,E1 -354.698,E2 -354.698} C_VEL
LIN {X 0,Y 608.478,Z 379.689,A -85,B 0,C 180,E1 -357.352,E2 -357.352} C_VEL
LIN {X 0,Y 608.47,Z 379.691,A -85,B 0,C 180,E1 -360,E2 -360} C_VEL
LIN {X 0,Y 608.483,Z 379.693,A -85,B 0,C 180,E1 -362.648,E2 -362.648} C_VEL
LIN {X 0,Y 608.466,Z 379.693,A -85,B 0,C 180,E1 -365.302,E2 -365.302} C_VEL
LIN {X 0,Y 608.47,Z 379.69,A -85,B 0,C 180,E1 -367.967,E2 -367.967} C_VEL
LIN {X 0,Y 608.461,Z 379.691,A -85,B 0,C 180,E1 -370.65,E2 -370.65} C_VEL
LIN {X 0,Y 608.468,Z 379.692,A -85,B 0,C 180,E1 -373.356,E2 -373.356} C_VEL
LIN {X 0,Y 608.461,Z 379.696,A -85,B 0,C 180,E1 -376.094,E2 -376.094} C_VEL
LIN {X 0,Y 608.454,Z 379.697,A -85,B 0,C 180,E1 -378.87,E2 -378.87} C_VEL
LIN {X 0,Y 608.468,Z 379.693,A -85,B 0,C 180,E1 -381.692,E2 -381.692} C_VEL
LIN {X 0,Y 608.457,Z 379.693,A -85,B 0,C 180,E1 -384.571,E2 -384.571} C_VEL
LIN {X 0,Y 608.482,Z 379.688,A -85,B 0,C 180,E1 -387.21,E2 -387.21} C_VEL
LIN {X 0,Y 608.472,Z 379.69,A -85,B 0,C 180,E1 -389.974,E2 -389.974} C_VEL
LIN {X 0,Y 608.467,Z 379.695,A -85,B 0,C 180,E1 -392.525,E2 -392.525} C_VEL
LIN {X 0,Y 608.45,Z 379.697,A -85,B 0,C 180,E1 -395.277,E2 -395.277} C_VEL
LIN {X 0,Y 608.471,Z 379.694,A -85,B 0,C 180,E1 -398.242,E2 -398.242} C_VEL
LIN {X 0,Y 608.447,Z 379.694,A -85,B 0,C 180,E1 -400.33,E2 -400.33} C_VEL
LIN {X 0,Y 608.454,Z 379.697,A -85,B 0,C 180,E1 -402.96,E2 -402.96} C_VEL
LIN {X 0,Y 608.463,Z 379.695,A -85,B 0,C 180,E1 -405.736,E2 -405.736} C_VEL
LIN {X 0,Y 608.465,Z 379.694,A -85,B 0,C 180,E1 -408.658,E2 -408.658} C_VEL
LIN {X 0,Y 608.466,Z 379.692,A -85,B 0,C 180,E1 -411.413,E2 -411.413} C_VEL
LIN {X 0,Y 608.459,Z 379.692,A -85,B 0,C 180,E1 -413.953,E2 -413.953} C_VEL
LIN {X 0,Y 608.477,Z 379.8,A -85,B 0,C 180,E1 -414.472,E2 -414.472} C_VEL
LIN {X 0,Y 608.498,Z 387.16,A -85,B 0,C 180,E1 -417.124,E2 -417.124} C_VEL
LIN {X 0,Y 608.482,Z 395.506,A -85,B 0,C 180,E1 -420.027,E2 -420.027} C_VEL
LIN {X 0,Y 608.474,Z 403.681,A -85,B 0,C 180,E1 -422.794,E2 -422.794} C_VEL
LIN {X 0,Y 608.466,Z 411.658,A -85,B 0,C 180,E1 -425.43,E2 -425.43} C_VEL
LIN {X 0,Y 608.453,Z 420.562,A -85,B 0,C 180,E1 -428.308,E2 -428.308} C_VEL
LIN {X 0,Y 608.46,Z 429.466,A -85,B 0,C 180,E1 -431.131,E2 -431.131} C_VEL
LIN {X 0,Y 608.442,Z 438.37,A -85,B 0,C 180,E1 -433.906,E2 -433.906} C_VEL
LIN {X 0,Y 608.438,Z 447.275,A -85,B 0,C 180,E1 -436.643,E2 -436.643} C_VEL
LIN {X 0,Y 608.436,Z 452.492,A -85,B 0,C 180,E1 -438.232,E2 -438.232} C_VEL
LIN {X 0,Y 608.544,Z 466.701,A -85,B 0,C 180,E1 -438.53,E2 -438.53} C_VEL
LIN {X 0,Y 608.521,Z 479.468,A -85,B 0,C 180,E1 -438.939,E2 -438.939} C_VEL
LIN {X 0,Y 608.51,Z 490.923,A -85,B 0,C 180,E1 -439.435,E2 -439.435} C_VEL
LIN {X 0,Y 608.489,Z 501.58,A -85,B 0,C 180,E1 -440.023,E2 -440.023} C_VEL
LIN {X 0,Y 608.483,Z 512.475,A -85,B 0,C 180,E1 -440.778,E2 -440.778} C_VEL
LIN {X 0,Y 608.475,Z 523.112,A -85,B 0,C 180,E1 -441.699,E2 -441.699} C_VEL
LIN {X 0,Y 608.471,Z 530.961,A -85,B 0,C 180,E1 -442.534,E2 -442.534} C_VEL
LIN {X 0,Y 608.461,Z 538.287,A -85,B 0,C 180,E1 -443.485,E2 -443.485} C_VEL
LIN {X 0,Y 608.45,Z 543.866,A -85,B 0,C 180,E1 -444.366,E2 -444.366} C_VEL
LIN {X 0,Y 608.432,Z 548.95,A -85,B 0,C 180,E1 -445.362,E2 -445.362} C_VEL
LIN {X 0,Y 608.449,Z 552.896,A -85,B 0,C 180,E1 -446.358,E2 -446.358} C_VEL
LIN {X 0,Y 608.425,Z 555.809,A -85,B 0,C 180,E1 -447.352,E2 -447.352} C_VEL
LIN {X 0,Y 608.444,Z 557.201,A -85,B 0,C 180,E1 -448.014,E2 -448.014} C_VEL
LIN {X 0,Y 608.438,Z 558.783,A -85,B 0,C 180,E1 -449.338,E2 -449.338} C_VEL
LIN {X 0,Y 608.434,Z 559,A -85,B 0,C 180,E1 -450,E2 -450} C_VEL
LIN {X 0,Y 608.448,Z 558.184,A -85,B 0,C 180,E1 -451.324,E2 -451.324} C_VEL
LIN {X 0,Y 608.444,Z 557.202,A -85,B 0,C 180,E1 -451.986,E2 -451.986} C_VEL
LIN {X 0,Y 608.425,Z 555.81,A -85,B 0,C 180,E1 -452.648,E2 -452.648} C_VEL
LIN {X 0,Y 608.449,Z 552.897,A -85,B 0,C 180,E1 -453.642,E2 -453.642} C_VEL
LIN {X 0,Y 608.432,Z 548.951,A -85,B 0,C 180,E1 -454.638,E2 -454.638} C_VEL
LIN {X 0,Y 608.437,Z 542.878,A -85,B 0,C 180,E1 -455.801,E2 -455.801} C_VEL
LIN {X 0,Y 608.462,Z 536.237,A -85,B 0,C 180,E1 -456.799,E2 -456.799} C_VEL
LIN {X 0,Y 608.455,Z 527.992,A -85,B 0,C 180,E1 -457.8,E2 -457.8} C_VEL
LIN {X 0,Y 608.472,Z 519.54,A -85,B 0,C 180,E1 -458.635,E2 -458.635} C_VEL
LIN {X 0,Y 608.481,Z 509.095,A -85,B 0,C 180,E1 -459.473,E2 -459.473} C_VEL
LIN {X 0,Y 608.491,Z 498.761,A -85,B 0,C 180,E1 -460.144,E2 -460.144} C_VEL
LIN {X 0,Y 608.517,Z 487.265,A -85,B 0,C 180,E1 -460.74,E2 -460.74} C_VEL
LIN {X 0,Y 608.537,Z 474.901,A -85,B 0,C 180,E1 -461.224,E2 -461.224} C_VEL
LIN {X 0,Y 608.546,Z 461.455,A -85,B 0,C 180,E1 -461.596,E2 -461.596} C_VEL
LIN {X 0,Y 608.436,Z 452.493,A -85,B 0,C 180,E1 -461.767,E2 -461.767} C_VEL
LIN {X 0,Y 608.424,Z 443.936,A -85,B 0,C 180,E1 -464.379,E2 -464.379} C_VEL
LIN {X 0,Y 608.451,Z 436.145,A -85,B 0,C 180,E1 -466.784,E2 -466.784} C_VEL
LIN {X 0,Y 608.457,Z 427.241,A -85,B 0,C 180,E1 -469.57,E2 -469.57} C_VEL
LIN {X 0,Y 608.478,Z 418.337,A -85,B 0,C 180,E1 -472.405,E2 -472.405} C_VEL
LIN {X 0,Y 608.465,Z 410.545,A -85,B 0,C 180,E1 -474.934,E2 -474.934} C_VEL
LIN {X 0,Y 608.473,Z 402.754,A -85,B 0,C 180,E1 -477.516,E2 -477.516} C_VEL
LIN {X 0,Y 608.484,Z 395.504,A -85,B 0,C 180,E1 -479.974,E2 -479.974} C_VEL
LIN {X 0,Y 608.498,Z 387.142,A -85,B 0,C 180,E1 -482.876,E2 -482.876} C_VEL
LIN {X 0,Y 608.486,Z 379.696,A -85,B 0,C 180,E1 -485.566,E2 -485.566} C_VEL
LIN {X 0,Y 608.465,Z 379.687,A -85,B 0,C 180,E1 -488.24,E2 -488.24} C_VEL
LIN {X 0,Y 608.452,Z 379.689,A -85,B 0,C 180,E1 -490.329,E2 -490.329} C_VEL
LIN {X 0,Y 608.482,Z 379.688,A -85,B 0,C 180,E1 -493.31,E2 -493.31} C_VEL
LIN {X 0,Y 608.47,Z 379.687,A -85,B 0,C 180,E1 -496.13,E2 -496.13} C_VEL
LIN {X 0,Y 608.462,Z 379.695,A -85,B 0,C 180,E1 -498.824,E2 -498.824} C_VEL
LIN {X 0,Y 608.469,Z 379.686,A -85,B 0,C 180,E1 -501.412,E2 -501.412} C_VEL
LIN {X 0,Y 608.475,Z 379.687,A -85,B 0,C 180,E1 -503.949,E2 -503.949} C_VEL
LIN {X 0,Y 608.468,Z 379.695,A -85,B 0,C 180,E1 -506.329,E2 -506.329} C_VEL
LIN {X 0,Y 608.472,Z 379.69,A -85,B 0,C 180,E1 -508.726,E2 -508.726} C_VEL
LIN {X 0,Y 608.466,Z 379.686,A -85,B 0,C 180,E1 -511.379,E2 -511.379} C_VEL
LIN {X 0,Y 608.437,Z 379.697,A -85,B 0,C 180,E1 -513.964,E2 -513.964} C_VEL
LIN {X 0,Y 608.468,Z 379.695,A -85,B 0,C 180,E1 -516.155,E2 -516.155} C_VEL
LIN {X 0,Y 608.448,Z 379.688,A -85,B 0,C 180,E1 -519.018,E2 -519.018} C_VEL
LIN {X 0,Y 608.444,Z 379.698,A -85,B 0,C 180,E1 -521.828,E2 -521.828} C_VEL
LIN {X 0,Y 608.47,Z 379.686,A -85,B 0,C 180,E1 -524.594,E2 -524.594} C_VEL
LIN {X 0,Y 608.474,Z 379.689,A -85,B 0,C 180,E1 -527.323,E2 -527.323} C_VEL
LIN {X 0,Y 608.449,Z 379.692,A -85,B 0,C 180,E1 -530.022,E2 -530.022} C_VEL
LIN {X 0,Y 608.478,Z 379.685,A -85,B 0,C 180,E1 -532.701,E2 -532.701} C_VEL
LIN {X 0,Y 608.467,Z 379.696,A -85,B 0,C 180,E1 -535.362,E2 -535.362} C_VEL
LIN {X 0,Y 608.449,Z 379.689,A -85,B 0,C 180,E1 -538.014,E2 -538.014} C_VEL
LIN {X 0,Y 608.477,Z 379.687,A -85,B 0,C 180,E1 -540.662,E2 -540.662} C_VEL
LIN {X 0,Y 608.487,Z 379.691,A -85,B 0,C 180,E1 -543.311,E2 -543.311} C_VEL
LIN {X 0,Y 608.452,Z 379.688,A -85,B 0,C 180,E1 -545.967,E2 -545.967} C_VEL
LIN {X 0,Y 608.456,Z 379.692,A -85,B 0,C 180,E1 -548.636,E2 -548.636} C_VEL
LIN {X 0,Y 608.461,Z 379.689,A -85,B 0,C 180,E1 -549.468,E2 -549.468} C_VEL
LIN {X 0,Y 607.774,Z 379.775,A -85,B 0,C 180,E1 -550.021,E2 -550.021} C_VEL
LIN {X 0,Y 604.913,Z 380.139,A -85,B 0,C 180,E1 -550.918,E2 -550.918} C_VEL
LIN {X 0,Y 602.512,Z 380.432,A -85,B 0,C 180,E1 -551.639,E2 -551.639} C_VEL
LIN {X 0,Y 601.487,Z 380.557,A -85,B 0,C 180,E1 -552.196,E2 -552.196} C_VEL
LIN {X 0,Y 601.406,Z 380.569,A -85,B 0,C 180,E1 -552.384,E2 -552.384} C_VEL
LIN {X 0,Y 601.428,Z 380.571,A -85,B 0,C 180,E1 -554.897,E2 -554.897} C_VEL
LIN {X 0,Y 601.431,Z 380.568,A -85,B 0,C 180,E1 -556.986,E2 -556.986} C_VEL
LIN {X 0,Y 601.407,Z 380.566,A -85,B 0,C 180,E1 -559.809,E2 -559.809} C_VEL
LIN {X 0,Y 601.447,Z 380.567,A -85,B 0,C 180,E1 -562.682,E2 -562.682} C_VEL
LIN {X 0,Y 601.404,Z 380.569,A -85,B 0,C 180,E1 -564.878,E2 -564.878} C_VEL
LIN {X 0,Y 601.42,Z 380.567,A -85,B 0,C 180,E1 -567.867,E2 -567.867} C_VEL
LIN {X 0,Y 601.441,Z 380.571,A -85,B 0,C 180,E1 -570.163,E2 -570.163} C_VEL
LIN {X 0,Y 601.419,Z 380.566,A -85,B 0,C 180,E1 -572.717,E2 -572.717} C_VEL
LIN {X 0,Y 601.411,Z 380.565,A -85,B 0,C 180,E1 -575.116,E2 -575.116} C_VEL
LIN {X 0,Y 601.429,Z 380.565,A -85,B 0,C 180,E1 -577.419,E2 -577.419} C_VEL
LIN {X 0,Y 601.408,Z 380.574,A -85,B 0,C 180,E1 -579.995,E2 -579.995} C_VEL
LIN {X 0,Y 601.406,Z 380.566,A -85,B 0,C 180,E1 -582.671,E2 -582.671} C_VEL
LIN {X 0,Y 601.42,Z 380.571,A -85,B 0,C 180,E1 -585.483,E2 -585.483} C_VEL
LIN {X 0,Y 601.424,Z 380.564,A -85,B 0,C 180,E1 -588.407,E2 -588.407} C_VEL
LIN {X 0,Y 601.432,Z 380.564,A -85,B 0,C 180,E1 -590.876,E2 -590.876} C_VEL
LIN {X 0,Y 601.44,Z 380.566,A -85,B 0,C 180,E1 -593.734,E2 -593.734} C_VEL
LIN {X 0,Y 601.432,Z 380.563,A -85,B 0,C 180,E1 -596.064,E2 -596.064} C_VEL
LIN {X 0,Y 601.441,Z 380.562,A -85,B 0,C 180,E1 -598.542,E2 -598.542} C_VEL
LIN {X 0,Y 601.436,Z 380.568,A -85,B 0,C 180,E1 -601.374,E2 -601.374} C_VEL
LIN {X 0,Y 601.405,Z 380.568,A -85,B 0,C 180,E1 -603.637,E2 -603.637} C_VEL
LIN {X 0,Y 601.422,Z 380.568,A -85,B 0,C 180,E1 -606.59,E2 -606.59} C_VEL
LIN {X 0,Y 601.381,Z 380.621,A -85,B 0,C 180,E1 -608.76,E2 -608.76} C_VEL
LIN {X 0,Y 601.406,Z 384.77,A -85,B 0,C 180,E1 -611.184,E2 -611.184} C_VEL
LIN {X 0,Y 601.374,Z 389.161,A -85,B 0,C 180,E1 -613.712,E2 -613.712} C_VEL
LIN {X 0,Y 601.379,Z 394.154,A -85,B 0,C 180,E1 -616.484,E2 -616.484} C_VEL
LIN {X 0,Y 601.385,Z 399.231,A -85,B 0,C 180,E1 -619.224,E2 -619.224} C_VEL
LIN {X 0,Y 601.387,Z 404.373,A -85,B 0,C 180,E1 -621.939,E2 -621.939} C_VEL
LIN {X 0,Y 601.369,Z 409.582,A -85,B 0,C 180,E1 -624.636,E2 -624.636} C_VEL
LIN {X 0,Y 601.33,Z 414.855,A -85,B 0,C 180,E1 -627.321,E2 -627.321} C_VEL
LIN {X 0,Y 601.351,Z 420.188,A -85,B 0,C 180,E1 -630,E2 -630} C_VEL
LIN {X 0,Y 601.379,Z 424.525,A -85,B 0,C 180,E1 -632.156,E2 -632.156} C_VEL
LIN {X 0,Y 601.629,Z 430.941,A -85,B 0,C 180,E1 -632.301,E2 -632.301} C_VEL
LIN {X 0,Y 601.557,Z 443.319,A -85,B 0,C 180,E1 -632.637,E2 -632.637} C_VEL
LIN {X 0,Y 601.519,Z 455.418,A -85,B 0,C 180,E1 -633.098,E2 -633.098} C_VEL
LIN {X 0,Y 601.519,Z 467.118,A -85,B 0,C 180,E1 -633.684,E2 -633.684} C_VEL
LIN {X 0,Y 601.469,Z 477.664,A -85,B 0,C 180,E1 -634.356,E2 -634.356} C_VEL
LIN {X 0,Y 601.431,Z 488.263,A -85,B 0,C 180,E1 -635.196,E2 -635.196} C_VEL
LIN {X 0,Y 601.405,Z 496.927,A -85,B 0,C 180,E1 -636.037,E2 -636.037} C_VEL
LIN {X 0,Y 601.382,Z 505.378,A -85,B 0,C 180,E1 -637.048,E2 -637.048} C_VEL
LIN {X 0,Y 601.364,Z 512.193,A -85,B 0,C 180,E1 -638.062,E2 -638.062} C_VEL
LIN {X 0,Y 601.348,Z 517.66,A -85,B 0,C 180,E1 -639.078,E2 -639.078} C_VEL
LIN {X 0,Y 601.337,Z 521.944,A -85,B 0,C 180,E1 -640.097,E2 -640.097} C_VEL
LIN {X 0,Y 601.352,Z 524.783,A -85,B 0,C 180,E1 -640.976,E2 -640.976} C_VEL
LIN {X 0,Y 601.342,Z 527.379,A -85,B 0,C 180,E1 -642.144,E2 -642.144} C_VEL
LIN {X 0,Y 601.324,Z 528.329,A -85,B 0,C 180,E1 -642.83,E2 -642.83} C_VEL
LIN {X 0,Y 601.349,Z 528.999,A -85,B 0,C 180,E1 -644.064,E2 -644.064} C_VEL
LIN {X 0,Y 601.314,Z 528.655,A -85,B 0,C 180,E1 -644.9,E2 -644.9} C_VEL
LIN {X 0,Y 601.324,Z 527.939,A -85,B 0,C 180,E1 -645.593,E2 -645.593} C_VEL
LIN {X 0,Y 601.322,Z 526.115,A -85,B 0,C 180,E1 -646.588,E2 -646.588} C_VEL
LIN {X 0,Y 601.327,Z 523.025,A -85,B 0,C 180,E1 -647.69,E2 -647.69} C_VEL
LIN {X 0,Y 601.349,Z 518.676,A -85,B 0,C 180,E1 -648.8,E2 -648.8} C_VEL
LIN {X 0,Y 601.369,Z 512.431,A -85,B 0,C 180,E1 -649.988,E2 -649.988} C_VEL
LIN {X 0,Y 601.378,Z 504.983,A -85,B 0,C 180,E1 -651.096,E2 -651.096} C_VEL
LIN {X 0,Y 601.386,Z 497.792,A -85,B 0,C 180,E1 -651.96,E2 -651.96} C_VEL
LIN {X 0,Y 601.419,Z 488.61,A -85,B 0,C 180,E1 -652.864,E2 -652.864} C_VEL
LIN {X 0,Y 601.463,Z 478.379,A -85,B 0,C 180,E1 -653.682,E2 -653.682} C_VEL
LIN {X 0,Y 601.483,Z 467.106,A -85,B 0,C 180,E1 -654.407,E2 -654.407} C_VEL
LIN {X 0,Y 601.522,Z 454.978,A -85,B 0,C 180,E1 -655.011,E2 -655.011} C_VEL
LIN {X 0,Y 601.541,Z 442.732,A -85,B 0,C 180,E1 -655.473,E2 -655.473} C_VEL
LIN {X 0,Y 601.599,Z 429.456,A -85,B 0,C 180,E1 -655.821,E2 -655.821} C_VEL
LIN {X 0,Y 601.354,Z 424.521,A -85,B 0,C 180,E1 -655.937,E2 -655.937} C_VEL
LIN {X 0,Y 601.337,Z 418.825,A -85,B 0,C 180,E1 -658.772,E2 -658.772} C_VEL
LIN {X 0,Y 601.344,Z 413.525,A -85,B 0,C 180,E1 -661.443,E2 -661.443} C_VEL
LIN {X 0,Y 601.336,Z 408.283,A -85,B 0,C 180,E1 -664.124,E2 -664.124} C_VEL
LIN {X 0,Y 601.357,Z 403.546,A -85,B 0,C 180,E1 -666.586,E2 -666.586} C_VEL
LIN {X 0,Y 601.375,Z 397.994,A -85,B 0,C 180,E1 -669.528,E2 -669.528} C_VEL
LIN {X 0,Y 601.375,Z 392.212,A -85,B 0,C 180,E1 -672.673,E2 -672.673} C_VEL
LIN {X 0,Y 601.421,Z 387.265,A -85,B 0,C 180,E1 -675.482,E2 -675.482} C_VEL
LIN {X 0,Y 601.423,Z 382.208,A -85,B 0,C 180,E1 -678.406,E2 -678.406} C_VEL
LIN {X 0,Y 601.358,Z 380.579,A -85,B 0,C 180,E1 -679.432,E2 -679.432} C_VEL
LIN {X 0,Y 601.419,Z 380.569,A -85,B 0,C 180,E1 -681.732,E2 -681.732} C_VEL
LIN {X 0,Y 601.406,Z 380.571,A -85,B 0,C 180,E1 -684.247,E2 -684.247} C_VEL
LIN {X 0,Y 601.423,Z 380.574,A -85,B 0,C 180,E1 -686.686,E2 -686.686} C_VEL
LIN {X 0,Y 601.429,Z 380.567,A -85,B 0,C 180,E1 -689.059,E2 -689.059} C_VEL
LIN {X 0,Y 601.431,Z 380.57,A -85,B 0,C 180,E1 -691.373,E2 -691.373} C_VEL
LIN {X 0,Y 601.403,Z 380.571,A -85,B 0,C 180,E1 -693.636,E2 -693.636} C_VEL
LIN {X 0,Y 601.418,Z 380.569,A -85,B 0,C 180,E1 -696.59,E2 -696.59} C_VEL
LIN {X 0,Y 601.426,Z 380.567,A -85,B 0,C 180,E1 -699.478,E2 -699.478} C_VEL
LIN {X 0,Y 601.398,Z 380.571,A -85,B 0,C 180,E1 -702.312,E2 -702.312} C_VEL
LIN {X 0,Y 601.415,Z 380.572,A -85,B 0,C 180,E1 -704.409,E2 -704.409} C_VEL
LIN {X 0,Y 601.423,Z 380.569,A -85,B 0,C 180,E1 -707.172,E2 -707.172} C_VEL
LIN {X 0,Y 601.428,Z 380.567,A -85,B 0,C 180,E1 -709.905,E2 -709.905} C_VEL
LIN {X 0,Y 601.449,Z 380.565,A -85,B 0,C 180,E1 -712.615,E2 -712.615} C_VEL
LIN {X 0,Y 601.423,Z 380.571,A -85,B 0,C 180,E1 -715.308,E2 -715.308} C_VEL
LIN {X 0,Y 601.434,Z 380.571,A -85,B 0,C 180,E1 -717.991,E2 -717.991} C_VEL
LIN {X 0,Y 601.453,Z 380.565,A -85,B 0,C 180,E1 -720.67,E2 -720.67} C_VEL
LIN {X 0,Y 601.429,Z 380.567,A -85,B 0,C 180,E1 -723.35,E2 -723.35} C_VEL
LIN {X 0,Y 601.41,Z 380.57,A -85,B 0,C 180,E1 -726.037,E2 -726.037} C_VEL
LIN {X 0,Y 601.437,Z 380.569,A -85,B 0,C 180,E1 -728.738,E2 -728.738} C_VEL
LIN {X 0,Y 601.431,Z 380.572,A -85,B 0,C 180,E1 -731.458,E2 -731.458} C_VEL
LIN {X 0,Y 601.413,Z 380.571,A -85,B 0,C 180,E1 -734.206,E2 -734.206} C_VEL
LIN {X 0,Y 601.429,Z 380.568,A -85,B 0,C 180,E1 -736.986,E2 -736.986} C_VEL
LIN {X 0,Y 601.408,Z 380.57,A -85,B 0,C 180,E1 -739.809,E2 -739.809} C_VEL
LIN {X 0,Y 601.406,Z 380.57,A -85,B 0,C 180,E1 -742.683,E2 -742.683} C_VEL
LIN {X 0,Y 601.402,Z 380.576,A -85,B 0,C 180,E1 -744.879,E2 -744.879} C_VEL
LIN {X 0,Y 601.419,Z 380.569,A -85,B 0,C 180,E1 -747.365,E2 -747.365} C_VEL
LIN {X 0,Y 601.444,Z 380.565,A -85,B 0,C 180,E1 -750.163,E2 -750.163} C_VEL
LIN {X 0,Y 601.425,Z 380.57,A -85,B 0,C 180,E1 -752.717,E2 -752.717} C_VEL
LIN {X 0,Y 601.416,Z 380.571,A -85,B 0,C 180,E1 -755.116,E2 -755.116} C_VEL
LIN {X 0,Y 601.432,Z 380.567,A -85,B 0,C 180,E1 -757.419,E2 -757.419} C_VEL
LIN {X 0,Y 601.408,Z 380.574,A -85,B 0,C 180,E1 -759.996,E2 -759.996} C_VEL
LIN {X 0,Y 601.409,Z 380.573,A -85,B 0,C 180,E1 -762.671,E2 -762.671} C_VEL
LIN {X 0,Y 601.423,Z 380.569,A -85,B 0,C 180,E1 -765.483,E2 -765.483} C_VEL
LIN {X 0,Y 601.426,Z 380.569,A -85,B 0,C 180,E1 -768.407,E2 -768.407} C_VEL
LIN {X 0,Y 601.434,Z 380.567,A -85,B 0,C 180,E1 -770.876,E2 -770.876} C_VEL
LIN {X 0,Y 601.432,Z 380.57,A -85,B 0,C 180,E1 -773.736,E2 -773.736} C_VEL
LIN {X 0,Y 601.457,Z 380.717,A -85,B 0,C 180,E1 -774.337,E2 -774.337} C_VEL
LIN {X 0,Y 601.525,Z 387.099,A -85,B 0,C 180,E1 -776.693,E2 -776.693} C_VEL
LIN {X 0,Y 601.486,Z 394.959,A -85,B 0,C 180,E1 -779.452,E2 -779.452} C_VEL
LIN {X 0,Y 601.452,Z 402.753,A -85,B 0,C 180,E1 -782.135,E2 -782.135} C_VEL
LIN {X 0,Y 601.424,Z 411.658,A -85,B 0,C 180,E1 -785.123,E2 -785.123} C_VEL
LIN {X 0,Y 601.419,Z 418.572,A -85,B 0,C 180,E1 -787.395,E2 -787.395} C_VEL
LIN {X 0,Y 601.41,Z 427.24,A -85,B 0,C 180,E1 -790.191,E2 -790.191} C_VEL
LIN {X 0,Y 601.372,Z 436.144,A -85,B 0,C 180,E1 -793.013,E2 -793.013} C_VEL
LIN {X 0,Y 601.361,Z 445.049,A -85,B 0,C 180,E1 -795.793,E2 -795.793} C_VEL
LIN {X 0,Y 601.38,Z 452.492,A -85,B 0,C 180,E1 -798.092,E2 -798.092} C_VEL
LIN {X 0,Y 601.619,Z 465.937,A -85,B 0,C 180,E1 -798.375,E2 -798.375} C_VEL
LIN {X 0,Y 601.55,Z 478.121,A -85,B 0,C 180,E1 -798.758,E2 -798.758} C_VEL
LIN {X 0,Y 601.513,Z 490.925,A -85,B 0,C 180,E1 -799.311,E2 -799.311} C_VEL
LIN {X 0,Y 601.477,Z 501.581,A -85,B 0,C 180,E1 -799.906,E2 -799.906} C_VEL
LIN {X 0,Y 601.449,Z 512.476,A -85,B 0,C 180,E1 -800.669,E2 -800.669} C_VEL
LIN {X 0,Y 601.429,Z 523.112,A -85,B 0,C 180,E1 -801.601,E2 -801.601} C_VEL
LIN {X 0,Y 601.418,Z 530.961,A -85,B 0,C 180,E1 -802.446,E2 -802.446} C_VEL
LIN {X 0,Y 601.37,Z 538.225,A -85,B 0,C 180,E1 -803.398,E2 -803.398} C_VEL
LIN {X 0,Y 601.372,Z 543.866,A -85,B 0,C 180,E1 -804.299,E2 -804.299} C_VEL
LIN {X 0,Y 601.336,Z 548.95,A -85,B 0,C 180,E1 -805.307,E2 -805.307} C_VEL
LIN {X 0,Y 601.367,Z 552.896,A -85,B 0,C 180,E1 -806.315,E2 -806.315} C_VEL
LIN {X 0,Y 601.325,Z 555.809,A -85,B 0,C 180,E1 -807.32,E2 -807.32} C_VEL
LIN {X 0,Y 601.343,Z 557.201,A -85,B 0,C 180,E1 -807.991,E2 -807.991} C_VEL
LIN {X 0,Y 601.339,Z 558.784,A -85,B 0,C 180,E1 -809.33,E2 -809.33} C_VEL
LIN {X 0,Y 601.335,Z 559,A -85,B 0,C 180,E1 -810,E2 -810} C_VEL
LIN {X 0,Y 601.348,Z 558.184,A -85,B 0,C 180,E1 -811.339,E2 -811.339} C_VEL
LIN {X 0,Y 601.343,Z 557.202,A -85,B 0,C 180,E1 -812.009,E2 -812.009} C_VEL
LIN {X 0,Y 601.325,Z 555.81,A -85,B 0,C 180,E1 -812.679,E2 -812.679} C_VEL
LIN {X 0,Y 601.367,Z 552.897,A -85,B 0,C 180,E1 -813.685,E2 -813.685} C_VEL
LIN {X 0,Y 601.336,Z 548.951,A -85,B 0,C 180,E1 -814.692,E2 -814.692} C_VEL
LIN {X 0,Y 601.372,Z 542.878,A -85,B 0,C 180,E1 -815.869,E2 -815.869} C_VEL
LIN {X 0,Y 601.381,Z 536.237,A -85,B 0,C 180,E1 -816.879,E2 -816.879} C_VEL
LIN {X 0,Y 601.4,Z 527.992,A -85,B 0,C 180,E1 -817.892,E2 -817.892} C_VEL
LIN {X 0,Y 601.436,Z 519.54,A -85,B 0,C 180,E1 -818.737,E2 -818.737} C_VEL
LIN {X 0,Y 601.451,Z 509.096,A -85,B 0,C 180,E1 -819.585,E2 -819.585} C_VEL
LIN {X 0,Y 601.469,Z 498.763,A -85,B 0,C 180,E1 -820.264,E2 -820.264} C_VEL
LIN {X 0,Y 601.538,Z 486.597,A -85,B 0,C 180,E1 -820.896,E2 -820.896} C_VEL
LIN {X 0,Y 601.57,Z 474.227,A -85,B 0,C 180,E1 -821.378,E2 -821.378} C_VEL
LIN {X 0,Y 601.61,Z 461.454,A -85,B 0,C 180,E1 -821.732,E2 -821.732} C_VEL
LIN {X 0,Y 601.38,Z 452.493,A -85,B 0,C 180,E1 -821.908,E2 -821.908} C_VEL
LIN {X 0,Y 601.364,Z 443.936,A -85,B 0,C 180,E1 -824.552,E2 -824.552} C_VEL
LIN {X 0,Y 601.39,Z 435.032,A -85,B 0,C 180,E1 -827.337,E2 -827.337} C_VEL
LIN {X 0,Y 601.395,Z 426.128,A -85,B 0,C 180,E1 -830.165,E2 -830.165} C_VEL
LIN {X 0,Y 601.423,Z 417.224,A -85,B 0,C 180,E1 -833.045,E2 -833.045} C_VEL
LIN {X 0,Y 601.439,Z 409.432,A -85,B 0,C 180,E1 -835.616,E2 -835.616} C_VEL
LIN {X 0,Y 601.457,Z 401.641,A -85,B 0,C 180,E1 -838.244,E2 -838.244} C_VEL
LIN {X 0,Y 601.469,Z 393.807,A -85,B 0,C 180,E1 -840.938,E2 -840.938} C_VEL
LIN {X 0,Y 601.523,Z 385.35,A -85,B 0,C 180,E1 -843.948,E2 -843.948} C_VEL
LIN {X 0,Y 601.428,Z 380.568,A -85,B 0,C 180,E1 -845.751,E2 -845.751} C_VEL
LIN {X 0,Y 601.434,Z 380.565,A -85,B 0,C 180,E1 -848.471,E2 -848.471} C_VEL
LIN {X 0,Y 601.42,Z 380.573,A -85,B 0,C 180,E1 -850.873,E2 -850.873} C_VEL
LIN {X 0,Y 601.446,Z 380.562,A -85,B 0,C 180,E1 -853.583,E2 -853.583} C_VEL
LIN {X 0,Y 601.446,Z 380.565,A -85,B 0,C 180,E1 -856.424,E2 -856.424} C_VEL
LIN {X 0,Y 601.414,Z 380.565,A -85,B 0,C 180,E1 -859.425,E2 -859.425} C_VEL
LIN {X 0,Y 601.42,Z 380.564,A -85,B 0,C 180,E1 -861.732,E2 -861.732} C_VEL
LIN {X 0,Y 601.409,Z 380.571,A -85,B 0,C 180,E1 -864.247,E2 -864.247} C_VEL
LIN {X 0,Y 601.426,Z 380.569,A -85,B 0,C 180,E1 -866.686,E2 -866.686} C_VEL
LIN {X 0,Y 601.427,Z 380.564,A -85,B 0,C 180,E1 -869.058,E2 -869.058} C_VEL
LIN {X 0,Y 601.425,Z 380.563,A -85,B 0,C 180,E1 -871.373,E2 -871.373} C_VEL
LIN {X 0,Y 601.399,Z 380.569,A -85,B 0,C 180,E1 -873.636,E2 -873.636} C_VEL
LIN {X 0,Y 601.416,Z 380.567,A -85,B 0,C 180,E1 -876.589,E2 -876.589} C_VEL
LIN {X 0,Y 601.425,Z 380.566,A -85,B 0,C 180,E1 -879.478,E2 -879.478} C_VEL
LIN {X 0,Y 601.396,Z 380.57,A -85,B 0,C 180,E1 -882.311,E2 -882.311} C_VEL
LIN {X 0,Y 601.412,Z 380.567,A -85,B 0,C 180,E1 -884.409,E2 -884.409} C_VEL
LIN {X 0,Y 601.421,Z 380.566,A -85,B 0,C 180,E1 -887.172,E2 -887.172} C_VEL
LIN {X 0,Y 601.427,Z 380.569,A -85,B 0,C 180,E1 -889.905,E2 -889.905} C_VEL
LIN {X 0,Y 601.446,Z 380.561,A -85,B 0,C 180,E1 -892.615,E2 -892.615} C_VEL
LIN {X 0,Y 601.433,Z 380.571,A -85,B 0,C 180,E1 -895.308,E2 -895.308} C_VEL
LIN {X 0,Y 601.419,Z 380.565,A -85,B 0,C 180,E1 -897.991,E2 -897.991} C_VEL
LIN {X 0,Y 601.448,Z 380.563,A -85,B 0,C 180,E1 -900.669,E2 -900.669} C_VEL
LIN {X 0,Y 601.438,Z 380.569,A -85,B 0,C 180,E1 -903.349,E2 -903.349} C_VEL
LIN {X 0,Y 601.405,Z 380.566,A -85,B 0,C 180,E1 -906.037,E2 -906.037} C_VEL
LIN {X 0,Y 601.436,Z 380.569,A -85,B 0,C 180,E1 -908.738,E2 -908.738} C_VEL
LIN {X 0,Y 601.43,Z 380.564,A -85,B 0,C 180,E1 -911.458,E2 -911.458} C_VEL
LIN {X 0,Y 601.406,Z 380.569,A -85,B 0,C 180,E1 -912.384,E2 -912.384} C_VEL
LIN {X 0,Y 600.745,Z 380.657,A -85,B 0,C 180,E1 -912.944,E2 -912.944} C_VEL
LIN {X 0,Y 597.895,Z 381.013,A -85,B 0,C 180,E1 -913.851,E2 -913.851} C_VEL
LIN {X 0,Y 595.483,Z 381.311,A -85,B 0,C 180,E1 -914.581,E2 -914.581} C_VEL
LIN {X 0,Y 594.445,Z 381.437,A -85,B 0,C 180,E1 -915.145,E2 -915.145} C_VEL
LIN {X 0,Y 594.359,Z 381.445,A -85,B 0,C 180,E1 -915.336,E2 -915.336} C_VEL
LIN {X 0,Y 594.377,Z 381.442,A -85,B 0,C 180,E1 -917.904,E2 -917.904} C_VEL
LIN {X 0,Y 594.378,Z 381.445,A -85,B 0,C 180,E1 -920.919,E2 -920.919} C_VEL
LIN {X 0,Y 594.39,Z 381.441,A -85,B 0,C 180,E1 -923.704,E2 -923.704} C_VEL
LIN {X 0,Y 594.387,Z 381.444,A -85,B 0,C 180,E1 -926.699,E2 -926.699} C_VEL
LIN {X 0,Y 594.378,Z 381.442,A -85,B 0,C 180,E1 -928.999,E2 -928.999} C_VEL
LIN {X 0,Y 594.387,Z 381.443,A -85,B 0,C 180,E1 -931.646,E2 -931.646} C_VEL
LIN {X 0,Y 594.393,Z 381.442,A -85,B 0,C 180,E1 -934.579,E2 -934.579} C_VEL
LIN {X 0,Y 594.381,Z 381.441,A -85,B 0,C 180,E1 -937.087,E2 -937.087} C_VEL
LIN {X 0,Y 594.373,Z 381.45,A -85,B 0,C 180,E1 -939.776,E2 -939.776} C_VEL
LIN {X 0,Y 594.363,Z 381.445,A -85,B 0,C 180,E1 -942.376,E2 -942.376} C_VEL
LIN {X 0,Y 594.357,Z 381.446,A -85,B 0,C 180,E1 -945.192,E2 -945.192} C_VEL
LIN {X 0,Y 594.384,Z 381.45,A -85,B 0,C 180,E1 -947.627,E2 -947.627} C_VEL
LIN {X 0,Y 594.387,Z 381.44,A -85,B 0,C 180,E1 -950.322,E2 -950.322} C_VEL
LIN {X 0,Y 594.383,Z 381.443,A -85,B 0,C 180,E1 -952.914,E2 -952.914} C_VEL
LIN {X 0,Y 594.383,Z 381.443,A -85,B 0,C 180,E1 -955.861,E2 -955.861} C_VEL
LIN {X 0,Y 594.389,Z 381.442,A -85,B 0,C 180,E1 -958.652,E2 -958.652} C_VEL
LIN {X 0,Y 594.384,Z 381.449,A -85,B 0,C 180,E1 -961.042,E2 -961.042} C_VEL
LIN {X 0,Y 594.389,Z 381.44,A -85,B 0,C 180,E1 -963.977,E2 -963.977} C_VEL
LIN {X 0,Y 594.389,Z 381.441,A -85,B 0,C 180,E1 -966.297,E2 -966.297} C_VEL
LIN {X 0,Y 594.353,Z 381.448,A -85,B 0,C 180,E1 -968.497,E2 -968.497} C_VEL
LIN {X 0,Y 594.381,Z 382.224,A -85,B 0,C 180,E1 -969.224,E2 -969.224} C_VEL
LIN {X 0,Y 594.353,Z 387.116,A -85,B 0,C 180,E1 -972.095,E2 -972.095} C_VEL
LIN {X 0,Y 594.305,Z 392.008,A -85,B 0,C 180,E1 -974.921,E2 -974.921} C_VEL
LIN {X 0,Y 594.304,Z 397.03,A -85,B 0,C 180,E1 -977.71,E2 -977.71} C_VEL
LIN {X 0,Y 594.326,Z 400.853,A -85,B 0,C 180,E1 -979.783,E2 -979.783} C_VEL
LIN {X 0,Y 594.291,Z 406.011,A -85,B 0,C 180,E1 -982.526,E2 -982.526} C_VEL
LIN {X 0,Y 594.32,Z 411.231,A -85,B 0,C 180,E1 -985.252,E2 -985.252} C_VEL
LIN {X 0,Y 594.262,Z 416.52,A -85,B 0,C 180,E1 -987.967,E2 -987.967} C_VEL
LIN {X 0,Y 594.261,Z 421.87,A -85,B 0,C 180,E1 -990.678,E2 -990.678} C_VEL
LIN {X 0,Y 594.283,Z 424.525,A -85,B 0,C 180,E1 -992.012,E2 -992.012} C_VEL
LIN {X 0,Y 594.671,Z 429.872,A -85,B 0,C 180,E1 -992.138,E2 -992.138} C_VEL
LIN {X 0,Y 594.589,Z 441.956,A -85,B 0,C 180,E1 -992.456,E2 -992.456} C_VEL
LIN {X 0,Y 594.551,Z 453.409,A -85,B 0,C 180,E1 -992.88,E2 -992.88} C_VEL
LIN {X 0,Y 594.502,Z 465.536,A -85,B 0,C 180,E1 -993.474,E2 -993.474} C_VEL
LIN {X 0,Y 594.455,Z 476.434,A -85,B 0,C 180,E1 -994.153,E2 -994.153} C_VEL
LIN {X 0,Y 594.418,Z 486.301,A -85,B 0,C 180,E1 -994.917,E2 -994.917} C_VEL
LIN {X 0,Y 594.344,Z 495.285,A -85,B 0,C 180,E1 -995.769,E2 -995.769} C_VEL
LIN {X 0,Y 594.321,Z 504.083,A -85,B 0,C 180,E1 -996.791,E2 -996.791} C_VEL
LIN {X 0,Y 594.298,Z 511.16,A -85,B 0,C 180,E1 -997.816,E2 -997.816} C_VEL
LIN {X 0,Y 594.292,Z 516.828,A -85,B 0,C 180,E1 -998.843,E2 -998.843} C_VEL
LIN {X 0,Y 594.257,Z 521.306,A -85,B 0,C 180,E1 -999.874,E2 -999.874} C_VEL
LIN {X 0,Y 594.262,Z 524.969,A -85,B 0,C 180,E1 -1001.01,E2 -1001.01} C_VEL
LIN {X 0,Y 594.239,Z 527.656,A -85,B 0,C 180,E1 -1002.291,E2 -1002.291} C_VEL
LIN {X 0,Y 594.243,Z 528.516,A -85,B 0,C 180,E1 -1002.986,E2 -1002.986} C_VEL
LIN {X 0,Y 594.26,Z 528.988,A -85,B 0,C 180,E1 -1004.124,E2 -1004.124} C_VEL
LIN {X 0,Y 594.209,Z 528.534,A -85,B 0,C 180,E1 -1005.082,E2 -1005.082} C_VEL
LIN {X 0,Y 594.222,Z 527.678,A -85,B 0,C 180,E1 -1005.785,E2 -1005.785} C_VEL
LIN {X 0,Y 594.237,Z 526.008,A -85,B 0,C 180,E1 -1006.668,E2 -1006.668} C_VEL
LIN {X 0,Y 594.241,Z 522.426,A -85,B 0,C 180,E1 -1007.908,E2 -1007.908} C_VEL
LIN {X 0,Y 594.28,Z 517.631,A -85,B 0,C 180,E1 -1009.078,E2 -1009.078} C_VEL
LIN {X 0,Y 594.298,Z 511.381,A -85,B 0,C 180,E1 -1010.237,E2 -1010.237} C_VEL
LIN {X 0,Y 594.31,Z 505.074,A -85,B 0,C 180,E1 -1011.167,E2 -1011.167} C_VEL
LIN {X 0,Y 594.343,Z 497.82,A -85,B 0,C 180,E1 -1012.051,E2 -1012.051} C_VEL
LIN {X 0,Y 594.396,Z 488.649,A -85,B 0,C 180,E1 -1012.966,E2 -1012.966} C_VEL
LIN {X 0,Y 594.435,Z 478.419,A -85,B 0,C 180,E1 -1013.794,E2 -1013.794} C_VEL
LIN {X 0,Y 594.488,Z 467.341,A -85,B 0,C 180,E1 -1014.517,E2 -1014.517} C_VEL
LIN {X 0,Y 594.542,Z 455.162,A -85,B 0,C 180,E1 -1015.134,E2 -1015.134} C_VEL
LIN {X 0,Y 594.587,Z 442.845,A -85,B 0,C 180,E1 -1015.605,E2 -1015.605} C_VEL
LIN {X 0,Y 594.661,Z 429.665,A -85,B 0,C 180,E1 -1015.957,E2 -1015.957} C_VEL
LIN {X 0,Y 594.248,Z 424.544,A -85,B 0,C 180,E1 -1016.069,E2 -1016.069} C_VEL
LIN {X 0,Y 594.251,Z 418.858,A -85,B 0,C 180,E1 -1018.935,E2 -1018.935} C_VEL
LIN {X 0,Y 594.257,Z 413.59,A -85,B 0,C 180,E1 -1021.624,E2 -1021.624} C_VEL
LIN {X 0,Y 594.259,Z 408.766,A -85,B 0,C 180,E1 -1024.121,E2 -1024.121} C_VEL
LIN {X 0,Y 594.291,Z 403.124,A -85,B 0,C 180,E1 -1027.093,E2 -1027.093} C_VEL
LIN {X 0,Y 594.29,Z 398.159,A -85,B 0,C 180,E1 -1029.764,E2 -1029.764} C_VEL
LIN {X 0,Y 594.292,Z 393.404,A -85,B 0,C 180,E1 -1032.381,E2 -1032.381} C_VEL
LIN {X 0,Y 594.345,Z 389.218,A -85,B 0,C 180,E1 -1034.807,E2 -1034.807} C_VEL
LIN {X 0,Y 594.354,Z 384.358,A -85,B 0,C 180,E1 -1037.623,E2 -1037.623} C_VEL
LIN {X 0,Y 594.312,Z 381.457,A -85,B 0,C 180,E1 -1039.428,E2 -1039.428} C_VEL
LIN {X 0,Y 594.383,Z 381.449,A -85,B 0,C 180,E1 -1042.059,E2 -1042.059} C_VEL
LIN {X 0,Y 594.382,Z 381.446,A -85,B 0,C 180,E1 -1044.671,E2 -1044.671} C_VEL
LIN {X 0,Y 594.373,Z 381.448,A -85,B 0,C 180,E1 -1047.088,E2 -1047.088} C_VEL
LIN {X 0,Y 594.395,Z 381.449,A -85,B 0,C 180,E1 -1049.669,E2 -1049.669} C_VEL
LIN {X 0,Y 594.385,Z 381.449,A -85,B 0,C 180,E1 -1052.54,E2 -1052.54} C_VEL
LIN {X 0,Y 594.378,Z 381.445,A -85,B 0,C 180,E1 -1054.807,E2 -1054.807} C_VEL
LIN {X 0,Y 594.359,Z 381.452,A -85,B 0,C 180,E1 -1057.264,E2 -1057.264} C_VEL
LIN {X 0,Y 594.375,Z 381.449,A -85,B 0,C 180,E1 -1059.946,E2 -1059.946} C_VEL
LIN {X 0,Y 594.387,Z 381.446,A -85,B 0,C 180,E1 -1062.807,E2 -1062.807} C_VEL
LIN {X 0,Y 594.382,Z 381.447,A -85,B 0,C 180,E1 -1065.825,E2 -1065.825} C_VEL
LIN {X 0,Y 594.389,Z 381.444,A -85,B 0,C 180,E1 -1068.404,E2 -1068.404} C_VEL
LIN {X 0,Y 594.394,Z 381.444,A -85,B 0,C 180,E1 -1071.158,E2 -1071.158} C_VEL
LIN {X 0,Y 594.362,Z 381.449,A -85,B 0,C 180,E1 -1073.891,E2 -1073.891} C_VEL
LIN {X 0,Y 594.378,Z 381.451,A -85,B 0,C 180,E1 -1076.611,E2 -1076.611} C_VEL
LIN {X 0,Y 594.419,Z 381.443,A -85,B 0,C 180,E1 -1079.323,E2 -1079.323} C_VEL
LIN {X 0,Y 594.389,Z 381.445,A -85,B 0,C 180,E1 -1082.033,E2 -1082.033} C_VEL
LIN {X 0,Y 594.393,Z 381.443,A -85,B 0,C 180,E1 -1084.748,E2 -1084.748} C_VEL
LIN {X 0,Y 594.398,Z 381.443,A -85,B 0,C 180,E1 -1087.473,E2 -1087.473} C_VEL
LIN {X 0,Y 594.39,Z 381.447,A -85,B 0,C 180,E1 -1090.216,E2 -1090.216} C_VEL
LIN {X 0,Y 594.372,Z 381.452,A -85,B 0,C 180,E1 -1092.983,E2 -1092.983} C_VEL
LIN {X 0,Y 594.369,Z 381.45,A -85,B 0,C 180,E1 -1095.781,E2 -1095.781} C_VEL
LIN {X 0,Y 594.383,Z 381.447,A -85,B 0,C 180,E1 -1098.618,E2 -1098.618} C_VEL
LIN {X 0,Y 594.363,Z 381.448,A -85,B 0,C 180,E1 -1101.504,E2 -1101.504} C_VEL
LIN {X 0,Y 594.384,Z 381.445,A -85,B 0,C 180,E1 -1104.446,E2 -1104.446} C_VEL
LIN {X 0,Y 594.387,Z 381.447,A -85,B 0,C 180,E1 -1106.7,E2 -1106.7} C_VEL
LIN {X 0,Y 594.378,Z 381.446,A -85,B 0,C 180,E1 -1108.999,E2 -1108.999} C_VEL
LIN {X 0,Y 594.39,Z 381.444,A -85,B 0,C 180,E1 -1111.646,E2 -1111.646} C_VEL
LIN {X 0,Y 594.394,Z 381.443,A -85,B 0,C 180,E1 -1114.579,E2 -1114.579} C_VEL
LIN {X 0,Y 594.383,Z 381.448,A -85,B 0,C 180,E1 -1117.087,E2 -1117.087} C_VEL
LIN {X 0,Y 594.373,Z 381.45,A -85,B 0,C 180,E1 -1119.775,E2 -1119.775} C_VEL
LIN {X 0,Y 594.366,Z 381.448,A -85,B 0,C 180,E1 -1122.376,E2 -1122.376} C_VEL
LIN {X 0,Y 594.361,Z 381.448,A -85,B 0,C 180,E1 -1125.192,E2 -1125.192} C_VEL
LIN {X 0,Y 594.371,Z 381.449,A -85,B 0,C 180,E1 -1127.626,E2 -1127.626} C_VEL
LIN {X 0,Y 594.392,Z 381.449,A -85,B 0,C 180,E1 -1130.322,E2 -1130.322} C_VEL
LIN {X 0,Y 594.384,Z 381.447,A -85,B 0,C 180,E1 -1132.914,E2 -1132.914} C_VEL
LIN {X 0,Y 594.397,Z 381.587,A -85,B 0,C 180,E1 -1134.178,E2 -1134.178} C_VEL
LIN {X 0,Y 594.516,Z 385.992,A -85,B 0,C 180,E1 -1135.843,E2 -1135.843} C_VEL
LIN {X 0,Y 594.47,Z 392.869,A -85,B 0,C 180,E1 -1138.343,E2 -1138.343} C_VEL
LIN {X 0,Y 594.454,Z 400.597,A -85,B 0,C 180,E1 -1141.03,E2 -1141.03} C_VEL
LIN {X 0,Y 594.399,Z 407.205,A -85,B 0,C 180,E1 -1143.302,E2 -1143.302} C_VEL
LIN {X 0,Y 594.419,Z 415.011,A -85,B 0,C 180,E1 -1145.932,E2 -1145.932} C_VEL
LIN {X 0,Y 594.353,Z 424.609,A -85,B 0,C 180,E1 -1149.091,E2 -1149.091} C_VEL
LIN {X 0,Y 594.337,Z 432.805,A -85,B 0,C 180,E1 -1151.738,E2 -1151.738} C_VEL
LIN {X 0,Y 594.316,Z 441.71,A -85,B 0,C 180,E1 -1154.57,E2 -1154.57} C_VEL
LIN {X 0,Y 594.294,Z 451.727,A -85,B 0,C 180,E1 -1157.71,E2 -1157.71} C_VEL
LIN {X 0,Y 594.292,Z 452.492,A -85,B 0,C 180,E1 -1157.948,E2 -1157.948} C_VEL
LIN {X 0,Y 594.676,Z 457.236,A -85,B 0,C 180,E1 -1158.043,E2 -1158.043} C_VEL
LIN {X 0,Y 594.623,Z 470.5,A -85,B 0,C 180,E1 -1158.366,E2 -1158.366} C_VEL
LIN {X 0,Y 594.569,Z 482.173,A -85,B 0,C 180,E1 -1158.781,E2 -1158.781} C_VEL
LIN {X 0,Y 594.515,Z 494.211,A -85,B 0,C 180,E1 -1159.356,E2 -1159.356} C_VEL
LIN {X 0,Y 594.475,Z 505.478,A -85,B 0,C 180,E1 -1160.044,E2 -1160.044} C_VEL
LIN {X 0,Y 594.406,Z 515.647,A -85,B 0,C 180,E1 -1160.815,E2 -1160.815} C_VEL
LIN {X 0,Y 594.372,Z 524.788,A -85,B 0,C 180,E1 -1161.672,E2 -1161.672} C_VEL
LIN {X 0,Y 594.316,Z 533.691,A -85,B 0,C 180,E1 -1162.697,E2 -1162.697} C_VEL
LIN {X 0,Y 594.281,Z 540.169,A -85,B 0,C 180,E1 -1163.615,E2 -1163.615} C_VEL
LIN {X 0,Y 594.289,Z 545.68,A -85,B 0,C 180,E1 -1164.571,E2 -1164.571} C_VEL
LIN {X 0,Y 594.27,Z 550.371,A -85,B 0,C 180,E1 -1165.591,E2 -1165.591} C_VEL
LIN {X 0,Y 594.267,Z 553.956,A -85,B 0,C 180,E1 -1166.61,E2 -1166.61} C_VEL
LIN {X 0,Y 594.226,Z 555.809,A -85,B 0,C 180,E1 -1167.288,E2 -1167.288} C_VEL
LIN {X 0,Y 594.242,Z 557.201,A -85,B 0,C 180,E1 -1167.967,E2 -1167.967} C_VEL
LIN {X 0,Y 594.239,Z 558.784,A -85,B 0,C 180,E1 -1169.322,E2 -1169.322} C_VEL
LIN {X 0,Y 594.236,Z 559,A -85,B 0,C 180,E1 -1170,E2 -1170} C_VEL
LIN {X 0,Y 594.248,Z 558.185,A -85,B 0,C 180,E1 -1171.355,E2 -1171.355} C_VEL
LIN {X 0,Y 594.242,Z 557.202,A -85,B 0,C 180,E1 -1172.033,E2 -1172.033} C_VEL
LIN {X 0,Y 594.226,Z 555.81,A -85,B 0,C 180,E1 -1172.711,E2 -1172.711} C_VEL
LIN {X 0,Y 594.288,Z 552.897,A -85,B 0,C 180,E1 -1173.729,E2 -1173.729} C_VEL
LIN {X 0,Y 594.241,Z 548.951,A -85,B 0,C 180,E1 -1174.749,E2 -1174.749} C_VEL
LIN {X 0,Y 594.304,Z 542.879,A -85,B 0,C 180,E1 -1175.939,E2 -1175.939} C_VEL
LIN {X 0,Y 594.308,Z 536.238,A -85,B 0,C 180,E1 -1176.962,E2 -1176.962} C_VEL
LIN {X 0,Y 594.359,Z 527.992,A -85,B 0,C 180,E1 -1177.986,E2 -1177.986} C_VEL
LIN {X 0,Y 594.382,Z 519.54,A -85,B 0,C 180,E1 -1178.842,E2 -1178.842} C_VEL
LIN {X 0,Y 594.435,Z 509.098,A -85,B 0,C 180,E1 -1179.699,E2 -1179.699} C_VEL
LIN {X 0,Y 594.482,Z 498.764,A -85,B 0,C 180,E1 -1180.386,E2 -1180.386} C_VEL
LIN {X 0,Y 594.557,Z 487.734,A -85,B 0,C 180,E1 -1180.973,E2 -1180.973} C_VEL
LIN {X 0,Y 594.59,Z 475.723,A -85,B 0,C 180,E1 -1181.464,E2 -1181.464} C_VEL
LIN {X 0,Y 594.657,Z 462.367,A -85,B 0,C 180,E1 -1181.849,E2 -1181.849} C_VEL
LIN {X 0,Y 594.43,Z 453.639,A -85,B 0,C 180,E1 -1182.027,E2 -1182.027} C_VEL
LIN {X 0,Y 594.298,Z 452.423,A -85,B 0,C 180,E1 -1182.073,E2 -1182.073} C_VEL
LIN {X 0,Y 594.295,Z 442.823,A -85,B 0,C 180,E1 -1185.08,E2 -1185.08} C_VEL
LIN {X 0,Y 594.33,Z 433.919,A -85,B 0,C 180,E1 -1187.905,E2 -1187.905} C_VEL
LIN {X 0,Y 594.356,Z 425.015,A -85,B 0,C 180,E1 -1190.777,E2 -1190.777} C_VEL
LIN {X 0,Y 594.398,Z 416.111,A -85,B 0,C 180,E1 -1193.703,E2 -1193.703} C_VEL
LIN {X 0,Y 594.408,Z 409.182,A -85,B 0,C 180,E1 -1196.027,E2 -1196.027} C_VEL
LIN {X 0,Y 594.446,Z 401.676,A -85,B 0,C 180,E1 -1198.596,E2 -1198.596} C_VEL
LIN {X 0,Y 594.445,Z 393.749,A -85,B 0,C 180,E1 -1201.345,E2 -1201.345} C_VEL
LIN {X 0,Y 594.54,Z 385.99,A -85,B 0,C 180,E1 -1204.161,E2 -1204.161} C_VEL
LIN {X 0,Y 594.383,Z 381.446,A -85,B 0,C 180,E1 -1205.875,E2 -1205.875} C_VEL
LIN {X 0,Y 594.386,Z 381.447,A -85,B 0,C 180,E1 -1208.804,E2 -1208.804} C_VEL
LIN {X 0,Y 594.383,Z 381.441,A -85,B 0,C 180,E1 -1211.848,E2 -1211.848} C_VEL
LIN {X 0,Y 594.378,Z 381.443,A -85,B 0,C 180,E1 -1214.235,E2 -1214.235} C_VEL
LIN {X 0,Y 594.362,Z 381.447,A -85,B 0,C 180,E1 -1217.147,E2 -1217.147} C_VEL
LIN {X 0,Y 594.369,Z 381.443,A -85,B 0,C 180,E1 -1219.433,E2 -1219.433} C_VEL
LIN {X 0,Y 594.386,Z 381.447,A -85,B 0,C 180,E1 -1222.39,E2 -1222.39} C_VEL
LIN {X 0,Y 594.383,Z 381.448,A -85,B 0,C 180,E1 -1224.67,E2 -1224.67} C_VEL
LIN {X 0,Y 594.372,Z 381.443,A -85,B 0,C 180,E1 -1227.088,E2 -1227.088} C_VEL
LIN {X 0,Y 594.395,Z 381.441,A -85,B 0,C 180,E1 -1229.668,E2 -1229.668} C_VEL
LIN {X 0,Y 594.384,Z 381.445,A -85,B 0,C 180,E1 -1232.539,E2 -1232.539} C_VEL
LIN {X 0,Y 594.371,Z 381.443,A -85,B 0,C 180,E1 -1234.807,E2 -1234.807} C_VEL
LIN {X 0,Y 594.356,Z 381.445,A -85,B 0,C 180,E1 -1237.264,E2 -1237.264} C_VEL
LIN {X 0,Y 594.373,Z 381.452,A -85,B 0,C 180,E1 -1239.946,E2 -1239.946} C_VEL
LIN {X 0,Y 594.385,Z 381.441,A -85,B 0,C 180,E1 -1242.806,E2 -1242.806} C_VEL
LIN {X 0,Y 594.38,Z 381.45,A -85,B 0,C 180,E1 -1245.825,E2 -1245.825} C_VEL
LIN {X 0,Y 594.387,Z 381.441,A -85,B 0,C 180,E1 -1248.404,E2 -1248.404} C_VEL
LIN {X 0,Y 594.394,Z 381.443,A -85,B 0,C 180,E1 -1251.158,E2 -1251.158} C_VEL
LIN {X 0,Y 594.362,Z 381.447,A -85,B 0,C 180,E1 -1253.891,E2 -1253.891} C_VEL
LIN {X 0,Y 594.379,Z 381.442,A -85,B 0,C 180,E1 -1256.611,E2 -1256.611} C_VEL
LIN {X 0,Y 594.425,Z 381.445,A -85,B 0,C 180,E1 -1259.322,E2 -1259.322} C_VEL
LIN {X 0,Y 594.388,Z 381.44,A -85,B 0,C 180,E1 -1262.033,E2 -1262.033} C_VEL
LIN {X 0,Y 594.394,Z 381.444,A -85,B 0,C 180,E1 -1264.747,E2 -1264.747} C_VEL
LIN {X 0,Y 594.413,Z 381.44,A -85,B 0,C 180,E1 -1267.473,E2 -1267.473} C_VEL
LIN {X 0,Y 594.388,Z 381.441,A -85,B 0,C 180,E1 -1270.216,E2 -1270.216} C_VEL
LIN {X 0,Y 594.369,Z 381.45,A -85,B 0,C 180,E1 -1272.983,E2 -1272.983} C_VEL
LIN {X 0,Y 594.359,Z 381.445,A -85,B 0,C 180,E1 -1275.336,E2 -1275.336} C_VEL
LIN {X 0,Y 593.69,Z 381.528,A -85,B 0,C 180,E1 -1275.902,E2 -1275.902} C_VEL
LIN {X 0,Y 590.836,Z 381.89,A -85,B 0,C 180,E1 -1276.82,E2 -1276.82} C_VEL
LIN {X 0,Y 588.43,Z 382.188,A -85,B 0,C 180,E1 -1277.559,E2 -1277.559} C_VEL
LIN {X 0,Y 587.402,Z 382.313,A -85,B 0,C 180,E1 -1278.129,E2 -1278.129} C_VEL
LIN {X 0,Y 587.321,Z 382.323,A -85,B 0,C 180,E1 -1278.322,E2 -1278.322} C_VEL
LIN {X 0,Y 587.349,Z 382.32,A -85,B 0,C 180,E1 -1281.045,E2 -1281.045} C_VEL
LIN {X 0,Y 587.36,Z 382.316,A -85,B 0,C 180,E1 -1283.257,E2 -1283.257} C_VEL
LIN {X 0,Y 587.356,Z 382.325,A -85,B 0,C 180,E1 -1286.278,E2 -1286.278} C_VEL
LIN {X 0,Y 587.346,Z 382.318,A -85,B 0,C 180,E1 -1289.135,E2 -1289.135} C_VEL
LIN {X 0,Y 587.35,Z 382.322,A -85,B 0,C 180,E1 -1291.839,E2 -1291.839} C_VEL
LIN {X 0,Y 587.352,Z 382.322,A -85,B 0,C 180,E1 -1294.35,E2 -1294.35} C_VEL
LIN {X 0,Y 587.347,Z 382.318,A -85,B 0,C 180,E1 -1296.747,E2 -1296.747} C_VEL
LIN {X 0,Y 587.342,Z 382.32,A -85,B 0,C 180,E1 -1299.36,E2 -1299.36} C_VEL
LIN {X 0,Y 587.328,Z 382.324,A -85,B 0,C 180,E1 -1302.108,E2 -1302.108} C_VEL
LIN {X 0,Y 587.31,Z 382.323,A -85,B 0,C 180,E1 -1305.089,E2 -1305.089} C_VEL
LIN {X 0,Y 587.348,Z 382.322,A -85,B 0,C 180,E1 -1307.928,E2 -1307.928} C_VEL
LIN {X 0,Y 587.33,Z 382.322,A -85,B 0,C 180,E1 -1311.059,E2 -1311.059} C_VEL
LIN {X 0,Y 587.35,Z 382.324,A -85,B 0,C 180,E1 -1313.292,E2 -1313.292} C_VEL
LIN {X 0,Y 587.365,Z 382.318,A -85,B 0,C 180,E1 -1315.781,E2 -1315.781} C_VEL
LIN {X 0,Y 587.353,Z 382.316,A -85,B 0,C 180,E1 -1318.233,E2 -1318.233} C_VEL
LIN {X 0,Y 587.349,Z 382.322,A -85,B 0,C 180,E1 -1320.867,E2 -1320.867} C_VEL
LIN {X 0,Y 587.36,Z 382.316,A -85,B 0,C 180,E1 -1323.819,E2 -1323.819} C_VEL
LIN {X 0,Y 587.336,Z 382.319,A -85,B 0,C 180,E1 -1325.994,E2 -1325.994} C_VEL
LIN {X 0,Y 587.315,Z 382.322,A -85,B 0,C 180,E1 -1328.226,E2 -1328.226} C_VEL
LIN {X 0,Y 587.312,Z 382.621,A -85,B 0,C 180,E1 -1328.968,E2 -1328.968} C_VEL
LIN {X 0,Y 587.287,Z 387.521,A -85,B 0,C 180,E1 -1331.873,E2 -1331.873} C_VEL
LIN {X 0,Y 587.252,Z 392.454,A -85,B 0,C 180,E1 -1334.735,E2 -1334.735} C_VEL
LIN {X 0,Y 587.222,Z 397.376,A -85,B 0,C 180,E1 -1337.56,E2 -1337.56} C_VEL
LIN {X 0,Y 587.241,Z 401.196,A -85,B 0,C 180,E1 -1339.659,E2 -1339.659} C_VEL
LIN {X 0,Y 587.227,Z 406.351,A -85,B 0,C 180,E1 -1342.435,E2 -1342.435} C_VEL
LIN {X 0,Y 587.239,Z 411.571,A -85,B 0,C 180,E1 -1345.195,E2 -1345.195} C_VEL
LIN {X 0,Y 587.171,Z 416.859,A -85,B 0,C 180,E1 -1347.942,E2 -1347.942} C_VEL
LIN {X 0,Y 587.167,Z 422.209,A -85,B 0,C 180,E1 -1350.686,E2 -1350.686} C_VEL
LIN {X 0,Y 587.201,Z 424.526,A -85,B 0,C 180,E1 -1351.865,E2 -1351.865} C_VEL
LIN {X 0,Y 587.722,Z 429.715,A -85,B 0,C 180,E1 -1351.992,E2 -1351.992} C_VEL
LIN {X 0,Y 587.646,Z 441.848,A -85,B 0,C 180,E1 -1352.313,E2 -1352.313} C_VEL
LIN {X 0,Y 587.568,Z 453.342,A -85,B 0,C 180,E1 -1352.742,E2 -1352.742} C_VEL
LIN {X 0,Y 587.502,Z 465.488,A -85,B 0,C 180,E1 -1353.343,E2 -1353.343} C_VEL
LIN {X 0,Y 587.459,Z 476.388,A -85,B 0,C 180,E1 -1354.03,E2 -1354.03} C_VEL
LIN {X 0,Y 587.391,Z 486.268,A -85,B 0,C 180,E1 -1354.804,E2 -1354.804} C_VEL
LIN {X 0,Y 587.294,Z 495.259,A -85,B 0,C 180,E1 -1355.666,E2 -1355.666} C_VEL
LIN {X 0,Y 587.269,Z 503.623,A -85,B 0,C 180,E1 -1356.645,E2 -1356.645} C_VEL
LIN {X 0,Y 587.23,Z 511.142,A -85,B 0,C 180,E1 -1357.738,E2 -1357.738} C_VEL
LIN {X 0,Y 587.185,Z 517.63,A -85,B 0,C 180,E1 -1358.951,E2 -1358.951} C_VEL
LIN {X 0,Y 587.179,Z 521.92,A -85,B 0,C 180,E1 -1359.994,E2 -1359.994} C_VEL
LIN {X 0,Y 587.163,Z 525.142,A -85,B 0,C 180,E1 -1361.041,E2 -1361.041} C_VEL
LIN {X 0,Y 587.154,Z 526.743,A -85,B 0,C 180,E1 -1361.741,E2 -1361.741} C_VEL
LIN {X 0,Y 587.159,Z 527.917,A -85,B 0,C 180,E1 -1362.442,E2 -1362.442} C_VEL
LIN {X 0,Y 587.144,Z 528.639,A -85,B 0,C 180,E1 -1363.145,E2 -1363.145} C_VEL
LIN {X 0,Y 587.158,Z 528.976,A -85,B 0,C 180,E1 -1364.18,E2 -1364.18} C_VEL
LIN {X 0,Y 587.123,Z 528.353,A -85,B 0,C 180,E1 -1365.268,E2 -1365.268} C_VEL
LIN {X 0,Y 587.137,Z 527.399,A -85,B 0,C 180,E1 -1365.98,E2 -1365.98} C_VEL
LIN {X 0,Y 587.143,Z 525.907,A -85,B 0,C 180,E1 -1366.747,E2 -1366.747} C_VEL
LIN {X 0,Y 587.16,Z 523.046,A -85,B 0,C 180,E1 -1367.771,E2 -1367.771} C_VEL
LIN {X 0,Y 587.178,Z 518.314,A -85,B 0,C 180,E1 -1368.993,E2 -1368.993} C_VEL
LIN {X 0,Y 587.202,Z 512.467,A -85,B 0,C 180,E1 -1370.126,E2 -1370.126} C_VEL
LIN {X 0,Y 587.231,Z 505.281,A -85,B 0,C 180,E1 -1371.225,E2 -1371.225} C_VEL
LIN {X 0,Y 587.292,Z 497.847,A -85,B 0,C 180,E1 -1372.145,E2 -1372.145} C_VEL
LIN {X 0,Y 587.379,Z 487.901,A -85,B 0,C 180,E1 -1373.14,E2 -1373.14} C_VEL
LIN {X 0,Y 587.413,Z 477.195,A -85,B 0,C 180,E1 -1374.003,E2 -1374.003} C_VEL
LIN {X 0,Y 587.516,Z 466.688,A -85,B 0,C 180,E1 -1374.68,E2 -1374.68} C_VEL
LIN {X 0,Y 587.57,Z 454.068,A -85,B 0,C 180,E1 -1375.316,E2 -1375.316} C_VEL
LIN {X 0,Y 587.634,Z 441.685,A -85,B 0,C 180,E1 -1375.782,E2 -1375.782} C_VEL
LIN {X 0,Y 587.713,Z 429.234,A -85,B 0,C 180,E1 -1376.108,E2 -1376.108} C_VEL
LIN {X 0,Y 587.189,Z 424.517,A -85,B 0,C 180,E1 -1376.229,E2 -1376.229} C_VEL
LIN {X 0,Y 587.162,Z 418.893,A -85,B 0,C 180,E1 -1379.1,E2 -1379.1} C_VEL
LIN {X 0,Y 587.196,Z 413.647,A -85,B 0,C 180,E1 -1381.812,E2 -1381.812} C_VEL
LIN {X 0,Y 587.165,Z 408.866,A -85,B 0,C 180,E1 -1384.322,E2 -1384.322} C_VEL
LIN {X 0,Y 587.217,Z 404.295,A -85,B 0,C 180,E1 -1386.756,E2 -1386.756} C_VEL
LIN {X 0,Y 587.225,Z 399.483,A -85,B 0,C 180,E1 -1389.368,E2 -1389.368} C_VEL
LIN {X 0,Y 587.245,Z 394.635,A -85,B 0,C 180,E1 -1392.098,E2 -1392.098} C_VEL
LIN {X 0,Y 587.283,Z 389.498,A -85,B 0,C 180,E1 -1395.086,E2 -1395.086} C_VEL
LIN {X 0,Y 587.308,Z 384.642,A -85,B 0,C 180,E1 -1397.924,E2 -1397.924} C_VEL
LIN {X 0,Y 587.284,Z 382.96,A -85,B 0,C 180,E1 -1398.93,E2 -1398.93} C_VEL
LIN {X 0,Y 587.306,Z 382.327,A -85,B 0,C 180,E1 -1399.982,E2 -1399.982} C_VEL
LIN {X 0,Y 587.341,Z 382.326,A -85,B 0,C 180,E1 -1402.392,E2 -1402.392} C_VEL
LIN {X 0,Y 587.348,Z 382.325,A -85,B 0,C 180,E1 -1404.946,E2 -1404.946} C_VEL
LIN {X 0,Y 587.334,Z 382.323,A -85,B 0,C 180,E1 -1407.421,E2 -1407.421} C_VEL
LIN {X 0,Y 587.342,Z 382.326,A -85,B 0,C 180,E1 -1409.83,E2 -1409.83} C_VEL
LIN {X 0,Y 587.345,Z 382.323,A -85,B 0,C 180,E1 -1412.306,E2 -1412.306} C_VEL
LIN {X 0,Y 587.336,Z 382.325,A -85,B 0,C 180,E1 -1414.484,E2 -1414.484} C_VEL
LIN {X 0,Y 587.313,Z 382.331,A -85,B 0,C 180,E1 -1417.131,E2 -1417.131} C_VEL
LIN {X 0,Y 587.327,Z 382.325,A -85,B 0,C 180,E1 -1419.695,E2 -1419.695} C_VEL
LIN {X 0,Y 587.354,Z 382.321,A -85,B 0,C 180,E1 -1422.594,E2 -1422.594} C_VEL
LIN {X 0,Y 587.358,Z 382.321,A -85,B 0,C 180,E1 -1425.739,E2 -1425.739} C_VEL
LIN {X 0,Y 587.355,Z 382.323,A -85,B 0,C 180,E1 -1428.859,E2 -1428.859} C_VEL
LIN {X 0,Y 587.366,Z 382.321,A -85,B 0,C 180,E1 -1431.745,E2 -1431.745} C_VEL
LIN {X 0,Y 587.359,Z 382.32,A -85,B 0,C 180,E1 -1434.507,E2 -1434.507} C_VEL
LIN {X 0,Y 587.373,Z 382.318,A -85,B 0,C 180,E1 -1437.257,E2 -1437.257} C_VEL
LIN {X 0,Y 587.376,Z 382.319,A -85,B 0,C 180,E1 -1440,E2 -1440} C_VEL
LIN {X 0,Y 587.377,Z 382.321,A -85,B 0,C 180,E1 -1442.743,E2 -1442.743} C_VEL
LIN {X 0,Y 587.356,Z 382.325,A -85,B 0,C 180,E1 -1445.493,E2 -1445.493} C_VEL
LIN {X 0,Y 587.365,Z 382.321,A -85,B 0,C 180,E1 -1448.255,E2 -1448.255} C_VEL
LIN {X 0,Y 587.34,Z 382.324,A -85,B 0,C 180,E1 -1451.134,E2 -1451.134} C_VEL
LIN {X 0,Y 587.356,Z 382.32,A -85,B 0,C 180,E1 -1453.846,E2 -1453.846} C_VEL
LIN {X 0,Y 587.356,Z 382.32,A -85,B 0,C 180,E1 -1456.82,E2 -1456.82} C_VEL
LIN {X 0,Y 587.342,Z 382.322,A -85,B 0,C 180,E1 -1459.575,E2 -1459.575} C_VEL
LIN {X 0,Y 587.318,Z 382.328,A -85,B 0,C 180,E1 -1461.775,E2 -1461.775} C_VEL
LIN {X 0,Y 587.346,Z 382.325,A -85,B 0,C 180,E1 -1464.759,E2 -1464.759} C_VEL
LIN {X 0,Y 587.336,Z 382.323,A -85,B 0,C 180,E1 -1467.046,E2 -1467.046} C_VEL
LIN {X 0,Y 587.348,Z 382.326,A -85,B 0,C 180,E1 -1469.38,E2 -1469.38} C_VEL
LIN {X 0,Y 587.354,Z 382.321,A -85,B 0,C 180,E1 -1471.839,E2 -1471.839} C_VEL
LIN {X 0,Y 587.352,Z 382.322,A -85,B 0,C 180,E1 -1474.35,E2 -1474.35} C_VEL
LIN {X 0,Y 587.35,Z 382.324,A -85,B 0,C 180,E1 -1476.747,E2 -1476.747} C_VEL
LIN {X 0,Y 587.344,Z 382.322,A -85,B 0,C 180,E1 -1479.36,E2 -1479.36} C_VEL
LIN {X 0,Y 587.332,Z 382.323,A -85,B 0,C 180,E1 -1482.108,E2 -1482.108} C_VEL
LIN {X 0,Y 587.313,Z 382.326,A -85,B 0,C 180,E1 -1485.089,E2 -1485.089} C_VEL
LIN {X 0,Y 587.351,Z 382.321,A -85,B 0,C 180,E1 -1487.928,E2 -1487.928} C_VEL
LIN {X 0,Y 587.333,Z 382.324,A -85,B 0,C 180,E1 -1491.059,E2 -1491.059} C_VEL
LIN {X 0,Y 587.37,Z 382.41,A -85,B 0,C 180,E1 -1494,E2 -1494} C_VEL
LIN {X 0,Y 587.518,Z 387.084,A -85,B 0,C 180,E1 -1495.791,E2 -1495.791} C_VEL
LIN {X 0,Y 587.471,Z 393.692,A -85,B 0,C 180,E1 -1498.24,E2 -1498.24} C_VEL
LIN {X 0,Y 587.454,Z 401.126,A -85,B 0,C 180,E1 -1500.849,E2 -1500.849} C_VEL
LIN {X 0,Y 587.372,Z 409.704,A -85,B 0,C 180,E1 -1503.817,E2 -1503.817} C_VEL
LIN {X 0,Y 587.345,Z 417.223,A -85,B 0,C 180,E1 -1506.369,E2 -1506.369} C_VEL
LIN {X 0,Y 587.302,Z 426.142,A -85,B 0,C 180,E1 -1509.334,E2 -1509.334} C_VEL
LIN {X 0,Y 587.281,Z 435.031,A -85,B 0,C 180,E1 -1512.233,E2 -1512.233} C_VEL
LIN {X 0,Y 587.223,Z 443.936,A -85,B 0,C 180,E1 -1515.089,E2 -1515.089} C_VEL
LIN {X 0,Y 587.197,Z 452.492,A -85,B 0,C 180,E1 -1517.8,E2 -1517.8} C_VEL
LIN {X 0,Y 587.757,Z 457.236,A -85,B 0,C 180,E1 -1517.9,E2 -1517.9} C_VEL
LIN {X 0,Y 587.677,Z 470.501,A -85,B 0,C 180,E1 -1518.226,E2 -1518.226} C_VEL
LIN {X 0,Y 587.59,Z 483.177,A -85,B 0,C 180,E1 -1518.691,E2 -1518.691} C_VEL
LIN {X 0,Y 587.533,Z 494.212,A -85,B 0,C 180,E1 -1519.228,E2 -1519.228} C_VEL
LIN {X 0,Y 587.463,Z 505.479,A -85,B 0,C 180,E1 -1519.924,E2 -1519.924} C_VEL
LIN {X 0,Y 587.384,Z 515.648,A -85,B 0,C 180,E1 -1520.705,E2 -1520.705} C_VEL
LIN {X 0,Y 587.34,Z 524.788,A -85,B 0,C 180,E1 -1521.571,E2 -1521.571} C_VEL
LIN {X 0,Y 587.259,Z 533.691,A -85,B 0,C 180,E1 -1522.608,E2 -1522.608} C_VEL
LIN {X 0,Y 587.195,Z 540.746,A -85,B 0,C 180,E1 -1523.627,E2 -1523.627} C_VEL
LIN {X 0,Y 587.211,Z 545.68,A -85,B 0,C 180,E1 -1524.506,E2 -1524.506} C_VEL
LIN {X 0,Y 587.188,Z 550.371,A -85,B 0,C 180,E1 -1525.538,E2 -1525.538} C_VEL
LIN {X 0,Y 587.193,Z 553.956,A -85,B 0,C 180,E1 -1526.569,E2 -1526.569} C_VEL
LIN {X 0,Y 587.132,Z 555.808,A -85,B 0,C 180,E1 -1527.256,E2 -1527.256} C_VEL
LIN {X 0,Y 587.141,Z 557.2,A -85,B 0,C 180,E1 -1527.942,E2 -1527.942} C_VEL
LIN {X 0,Y 587.14,Z 558.784,A -85,B 0,C 180,E1 -1529.314,E2 -1529.314} C_VEL
LIN {X 0,Y 587.137,Z 559,A -85,B 0,C 180,E1 -1530,E2 -1530} C_VEL
LIN {X 0,Y 587.147,Z 558.185,A -85,B 0,C 180,E1 -1531.372,E2 -1531.372} C_VEL
LIN {X 0,Y 587.141,Z 557.201,A -85,B 0,C 180,E1 -1532.058,E2 -1532.058} C_VEL
LIN {X 0,Y 587.132,Z 555.81,A -85,B 0,C 180,E1 -1532.744,E2 -1532.744} C_VEL
LIN {X 0,Y 587.212,Z 552.897,A -85,B 0,C 180,E1 -1533.774,E2 -1533.774} C_VEL
LIN {X 0,Y 587.147,Z 548.95,A -85,B 0,C 180,E1 -1534.806,E2 -1534.806} C_VEL
LIN {X 0,Y 587.217,Z 542.879,A -85,B 0,C 180,E1 -1536.011,E2 -1536.011} C_VEL
LIN {X 0,Y 587.245,Z 536.238,A -85,B 0,C 180,E1 -1537.046,E2 -1537.046} C_VEL
LIN {X 0,Y 587.299,Z 527.992,A -85,B 0,C 180,E1 -1538.083,E2 -1538.083} C_VEL
LIN {X 0,Y 587.343,Z 519.541,A -85,B 0,C 180,E1 -1538.949,E2 -1538.949} C_VEL
LIN {X 0,Y 587.422,Z 509.099,A -85,B 0,C 180,E1 -1539.816,E2 -1539.816} C_VEL
LIN {X 0,Y 587.486,Z 498.764,A -85,B 0,C 180,E1 -1540.511,E2 -1540.511} C_VEL
LIN {X 0,Y 587.56,Z 486.822,A -85,B 0,C 180,E1 -1541.148,E2 -1541.148} C_VEL
LIN {X 0,Y 587.632,Z 474.609,A -85,B 0,C 180,E1 -1541.639,E2 -1541.639} C_VEL
LIN {X 0,Y 587.708,Z 461.452,A -85,B 0,C 180,E1 -1542.014,E2 -1542.014} C_VEL
LIN {X 0,Y 587.545,Z 454.671,A -85,B 0,C 180,E1 -1542.154,E2 -1542.154} C_VEL
LIN {X 0,Y 587.199,Z 452.423,A -85,B 0,C 180,E1 -1542.221,E2 -1542.221} C_VEL
LIN {X 0,Y 587.222,Z 443.936,A -85,B 0,C 180,E1 -1544.91,E2 -1544.91} C_VEL
LIN {X 0,Y 587.281,Z 435.032,A -85,B 0,C 180,E1 -1547.767,E2 -1547.767} C_VEL
LIN {X 0,Y 587.301,Z 426.143,A -85,B 0,C 180,E1 -1550.666,E2 -1550.666} C_VEL
LIN {X 0,Y 587.345,Z 417.224,A -85,B 0,C 180,E1 -1553.631,E2 -1553.631} C_VEL
LIN {X 0,Y 587.372,Z 409.432,A -85,B 0,C 180,E1 -1556.276,E2 -1556.276} C_VEL
LIN {X 0,Y 587.468,Z 400.45,A -85,B 0,C 180,E1 -1559.372,E2 -1559.372} C_VEL
LIN {X 0,Y 587.467,Z 393.468,A -85,B 0,C 180,E1 -1561.854,E2 -1561.854} C_VEL
LIN {X 0,Y 587.551,Z 386.638,A -85,B 0,C 180,E1 -1564.376,E2 -1564.376} C_VEL
LIN {X 0,Y 587.37,Z 382.322,A -85,B 0,C 180,E1 -1566.052,E2 -1566.052} C_VEL
LIN {X 0,Y 587.333,Z 382.328,A -85,B 0,C 180,E1 -1568.941,E2 -1568.941} C_VEL
LIN {X 0,Y 587.349,Z 382.317,A -85,B 0,C 180,E1 -1572.072,E2 -1572.072} C_VEL
LIN {X 0,Y 587.312,Z 382.327,A -85,B 0,C 180,E1 -1575.088,E2 -1575.088} C_VEL
LIN {X 0,Y 587.348,Z 382.318,A -85,B 0,C 180,E1 -1577.927,E2 -1577.927} C_VEL
LIN {X 0,Y 587.331,Z 382.322,A -85,B 0,C 180,E1 -1581.057,E2 -1581.057} C_VEL
LIN {X 0,Y 587.349,Z 382.318,A -85,B 0,C 180,E1 -1583.291,E2 -1583.291} C_VEL
LIN {X 0,Y 587.365,Z 382.316,A -85,B 0,C 180,E1 -1585.78,E2 -1585.78} C_VEL
LIN {X 0,Y 587.346,Z 382.325,A -85,B 0,C 180,E1 -1588.231,E2 -1588.231} C_VEL
LIN {X 0,Y 587.345,Z 382.319,A -85,B 0,C 180,E1 -1590.865,E2 -1590.865} C_VEL
LIN {X 0,Y 587.352,Z 382.321,A -85,B 0,C 180,E1 -1593.818,E2 -1593.818} C_VEL
LIN {X 0,Y 587.333,Z 382.327,A -85,B 0,C 180,E1 -1595.993,E2 -1595.993} C_VEL
LIN {X 0,Y 587.317,Z 382.328,A -85,B 0,C 180,E1 -1598.225,E2 -1598.225} C_VEL
LIN {X 0,Y 587.342,Z 382.319,A -85,B 0,C 180,E1 -1601.151,E2 -1601.151} C_VEL
LIN {X 0,Y 587.346,Z 382.32,A -85,B 0,C 180,E1 -1603.311,E2 -1603.311} C_VEL
LIN {X 0,Y 587.354,Z 382.32,A -85,B 0,C 180,E1 -1606.154,E2 -1606.154} C_VEL
LIN {X 0,Y 587.335,Z 382.32,A -85,B 0,C 180,E1 -1608.962,E2 -1608.962} C_VEL
LIN {X 0,Y 587.362,Z 382.322,A -85,B 0,C 180,E1 -1611.745,E2 -1611.745} C_VEL
LIN {X 0,Y 587.355,Z 382.317,A -85,B 0,C 180,E1 -1614.507,E2 -1614.507} C_VEL
LIN {X 0,Y 587.376,Z 382.322,A -85,B 0,C 180,E1 -1617.257,E2 -1617.257} C_VEL
LIN {X 0,Y 587.374,Z 382.315,A -85,B 0,C 180,E1 -1620,E2 -1620} C_VEL
LIN {X 0,Y 587.374,Z 382.318,A -85,B 0,C 180,E1 -1622.743,E2 -1622.743} C_VEL
LIN {X 0,Y 587.358,Z 382.32,A -85,B 0,C 180,E1 -1625.493,E2 -1625.493} C_VEL
LIN {X 0,Y 587.363,Z 382.316,A -85,B 0,C 180,E1 -1628.255,E2 -1628.255} C_VEL
LIN {X 0,Y 587.352,Z 382.322,A -85,B 0,C 180,E1 -1631.141,E2 -1631.141} C_VEL
LIN {X 0,Y 587.355,Z 382.319,A -85,B 0,C 180,E1 -1634.261,E2 -1634.261} C_VEL
LIN {X 0,Y 587.354,Z 382.317,A -85,B 0,C 180,E1 -1637.406,E2 -1637.406} C_VEL
LIN {X 0,Y 587.321,Z 382.323,A -85,B 0,C 180,E1 -1638.322,E2 -1638.322} C_VEL
LIN {X 0,Y 586.667,Z 382.408,A -85,B 0,C 180,E1 -1638.894,E2 -1638.894} C_VEL
LIN {X 0,Y 583.832,Z 382.759,A -85,B 0,C 180,E1 -1639.822,E2 -1639.822} C_VEL
LIN {X 0,Y 581.422,Z 383.065,A -85,B 0,C 180,E1 -1640.569,E2 -1640.569} C_VEL
LIN {X 0,Y 580.374,Z 383.188,A -85,B 0,C 180,E1 -1641.145,E2 -1641.145} C_VEL
LIN {X 0,Y 580.282,Z 383.198,A -85,B 0,C 180,E1 -1641.341,E2 -1641.341} C_VEL
LIN {X 0,Y 580.296,Z 383.196,A -85,B 0,C 180,E1 -1643.557,E2 -1643.557} C_VEL
LIN {X 0,Y 580.321,Z 383.202,A -85,B 0,C 180,E1 -1646.342,E2 -1646.342} C_VEL
LIN {X 0,Y 580.3,Z 383.195,A -85,B 0,C 180,E1 -1649.312,E2 -1649.312} C_VEL
LIN {X 0,Y 580.296,Z 383.204,A -85,B 0,C 180,E1 -1652.201,E2 -1652.201} C_VEL
LIN {X 0,Y 580.296,Z 383.197,A -85,B 0,C 180,E1 -1654.696,E2 -1654.696} C_VEL
LIN {X 0,Y 580.294,Z 383.197,A -85,B 0,C 180,E1 -1657.269,E2 -1657.269} C_VEL
LIN {X 0,Y 580.294,Z 383.199,A -85,B 0,C 180,E1 -1660.272,E2 -1660.272} C_VEL
LIN {X 0,Y 580.275,Z 383.198,A -85,B 0,C 180,E1 -1662.706,E2 -1662.706} C_VEL
LIN {X 0,Y 580.268,Z 383.208,A -85,B 0,C 180,E1 -1665.609,E2 -1665.609} C_VEL
LIN {X 0,Y 580.31,Z 383.195,A -85,B 0,C 180,E1 -1668.235,E2 -1668.235} C_VEL
LIN {X 0,Y 580.285,Z 383.199,A -85,B 0,C 180,E1 -1670.967,E2 -1670.967} C_VEL
LIN {X 0,Y 580.293,Z 383.202,A -85,B 0,C 180,E1 -1673.599,E2 -1673.599} C_VEL
LIN {X 0,Y 580.318,Z 383.193,A -85,B 0,C 180,E1 -1676.146,E2 -1676.146} C_VEL
LIN {X 0,Y 580.287,Z 383.198,A -85,B 0,C 180,E1 -1678.616,E2 -1678.616} C_VEL
LIN {X 0,Y 580.293,Z 383.204,A -85,B 0,C 180,E1 -1681.025,E2 -1681.025} C_VEL
LIN {X 0,Y 580.327,Z 383.193,A -85,B 0,C 180,E1 -1683.659,E2 -1683.659} C_VEL
LIN {X 0,Y 580.279,Z 383.2,A -85,B 0,C 180,E1 -1686.443,E2 -1686.443} C_VEL
LIN {X 0,Y 580.231,Z 383.27,A -85,B 0,C 180,E1 -1688.853,E2 -1688.853} C_VEL
LIN {X 0,Y 580.223,Z 387.93,A -85,B 0,C 180,E1 -1691.644,E2 -1691.644} C_VEL
LIN {X 0,Y 580.205,Z 391.621,A -85,B 0,C 180,E1 -1693.824,E2 -1693.824} C_VEL
LIN {X 0,Y 580.161,Z 396.538,A -85,B 0,C 180,E1 -1696.694,E2 -1696.694} C_VEL
LIN {X 0,Y 580.164,Z 401.54,A -85,B 0,C 180,E1 -1699.531,E2 -1699.531} C_VEL
LIN {X 0,Y 580.156,Z 406.692,A -85,B 0,C 180,E1 -1702.343,E2 -1702.343} C_VEL
LIN {X 0,Y 580.161,Z 411.91,A -85,B 0,C 180,E1 -1705.136,E2 -1705.136} C_VEL
LIN {X 0,Y 580.08,Z 417.198,A -85,B 0,C 180,E1 -1707.917,E2 -1707.917} C_VEL
LIN {X 0,Y 580.074,Z 422.547,A -85,B 0,C 180,E1 -1710.694,E2 -1710.694} C_VEL
LIN {X 0,Y 580.119,Z 424.526,A -85,B 0,C 180,E1 -1711.714,E2 -1711.714} C_VEL
LIN {X 0,Y 580.795,Z 430.519,A -85,B 0,C 180,E1 -1711.864,E2 -1711.864} C_VEL
LIN {X 0,Y 580.679,Z 443.034,A -85,B 0,C 180,E1 -1712.211,E2 -1712.211} C_VEL
LIN {X 0,Y 580.596,Z 455.212,A -85,B 0,C 180,E1 -1712.689,E2 -1712.689} C_VEL
LIN {X 0,Y 580.524,Z 466.97,A -85,B 0,C 180,E1 -1713.297,E2 -1713.297} C_VEL
LIN {X 0,Y 580.42,Z 477.546,A -85,B 0,C 180,E1 -1713.992,E2 -1713.992} C_VEL
LIN {X 0,Y 580.32,Z 488.174,A -85,B 0,C 180,E1 -1714.863,E2 -1714.863} C_VEL
LIN {X 0,Y 580.215,Z 496.857,A -85,B 0,C 180,E1 -1715.735,E2 -1715.735} C_VEL
LIN {X 0,Y 580.208,Z 504.419,A -85,B 0,C 180,E1 -1716.658,E2 -1716.658} C_VEL
LIN {X 0,Y 580.145,Z 511.127,A -85,B 0,C 180,E1 -1717.658,E2 -1717.658} C_VEL
LIN {X 0,Y 580.11,Z 516.802,A -85,B 0,C 180,E1 -1718.71,E2 -1718.71} C_VEL
LIN {X 0,Y 580.082,Z 521.283,A -85,B 0,C 180,E1 -1719.765,E2 -1719.765} C_VEL
LIN {X 0,Y 580.075,Z 525.329,A -85,B 0,C 180,E1 -1721.077,E2 -1721.077} C_VEL
LIN {X 0,Y 580.053,Z 527.078,A -85,B 0,C 180,E1 -1721.886,E2 -1721.886} C_VEL
LIN {X 0,Y 580.049,Z 528.119,A -85,B 0,C 180,E1 -1722.597,E2 -1722.597} C_VEL
LIN {X 0,Y 580.059,Z 528.757,A -85,B 0,C 180,E1 -1723.309,E2 -1723.309} C_VEL
LIN {X 0,Y 580.049,Z 528.964,A -85,B 0,C 180,E1 -1724.235,E2 -1724.235} C_VEL
LIN {X 0,Y 580.019,Z 528.155,A -85,B 0,C 180,E1 -1725.46,E2 -1725.46} C_VEL
LIN {X 0,Y 580.037,Z 527.114,A -85,B 0,C 180,E1 -1726.181,E2 -1726.181} C_VEL
LIN {X 0,Y 580.04,Z 525.602,A -85,B 0,C 180,E1 -1726.905,E2 -1726.905} C_VEL
LIN {X 0,Y 580.08,Z 522.452,A -85,B 0,C 180,E1 -1727.996,E2 -1727.996} C_VEL
LIN {X 0,Y 580.096,Z 518.13,A -85,B 0,C 180,E1 -1729.093,E2 -1729.093} C_VEL
LIN {X 0,Y 580.118,Z 512.484,A -85,B 0,C 180,E1 -1730.198,E2 -1730.198} C_VEL
LIN {X 0,Y 580.176,Z 505.305,A -85,B 0,C 180,E1 -1731.309,E2 -1731.309} C_VEL
LIN {X 0,Y 580.252,Z 497.875,A -85,B 0,C 180,E1 -1732.24,E2 -1732.24} C_VEL
LIN {X 0,Y 580.355,Z 488.347,A -85,B 0,C 180,E1 -1733.211,E2 -1733.211} C_VEL
LIN {X 0,Y 580.39,Z 478.497,A -85,B 0,C 180,E1 -1734.027,E2 -1734.027} C_VEL
LIN {X 0,Y 580.519,Z 467.325,A -85,B 0,C 180,E1 -1734.772,E2 -1734.772} C_VEL
LIN {X 0,Y 580.599,Z 455.215,A -85,B 0,C 180,E1 -1735.401,E2 -1735.401} C_VEL
LIN {X 0,Y 580.684,Z 442.402,A -85,B 0,C 180,E1 -1735.901,E2 -1735.901} C_VEL
LIN {X 0,Y 580.79,Z 429.454,A -85,B 0,C 180,E1 -1736.25,E2 -1736.25} C_VEL
LIN {X 0,Y 580.083,Z 424.512,A -85,B 0,C 180,E1 -1736.384,E2 -1736.384} C_VEL
LIN {X 0,Y 580.076,Z 418.93,A -85,B 0,C 180,E1 -1739.27,E2 -1739.27} C_VEL
LIN {X 0,Y 580.119,Z 413.316,A -85,B 0,C 180,E1 -1742.211,E2 -1742.211} C_VEL
LIN {X 0,Y 580.072,Z 408.624,A -85,B 0,C 180,E1 -1744.71,E2 -1744.71} C_VEL
LIN {X 0,Y 580.129,Z 403.872,A -85,B 0,C 180,E1 -1747.28,E2 -1747.28} C_VEL
LIN {X 0,Y 580.128,Z 399.063,A -85,B 0,C 180,E1 -1749.946,E2 -1749.946} C_VEL
LIN {X 0,Y 580.19,Z 394.34,A -85,B 0,C 180,E1 -1752.713,E2 -1752.713} C_VEL
LIN {X 0,Y 580.24,Z 389.776,A -85,B 0,C 180,E1 -1755.371,E2 -1755.371} C_VEL
LIN {X 0,Y 580.235,Z 384.95,A -85,B 0,C 180,E1 -1758.227,E2 -1758.227} C_VEL
LIN {X 0,Y 580.208,Z 383.446,A -85,B 0,C 180,E1 -1759.149,E2 -1759.149} C_VEL
LIN {X 0,Y 580.288,Z 383.204,A -85,B 0,C 180,E1 -1760.966,E2 -1760.966} C_VEL
LIN {X 0,Y 580.293,Z 383.205,A -85,B 0,C 180,E1 -1763.598,E2 -1763.598} C_VEL
LIN {X 0,Y 580.315,Z 383.198,A -85,B 0,C 180,E1 -1766.145,E2 -1766.145} C_VEL
LIN {X 0,Y 580.285,Z 383.202,A -85,B 0,C 180,E1 -1768.615,E2 -1768.615} C_VEL
LIN {X 0,Y 580.29,Z 383.204,A -85,B 0,C 180,E1 -1771.024,E2 -1771.024} C_VEL
LIN {X 0,Y 580.323,Z 383.197,A -85,B 0,C 180,E1 -1773.658,E2 -1773.658} C_VEL
LIN {X 0,Y 580.276,Z 383.202,A -85,B 0,C 180,E1 -1776.442,E2 -1776.442} C_VEL
LIN {X 0,Y 580.27,Z 383.203,A -85,B 0,C 180,E1 -1779.437,E2 -1779.437} C_VEL
LIN {X 0,Y 580.278,Z 383.208,A -85,B 0,C 180,E1 -1781.645,E2 -1781.645} C_VEL
LIN {X 0,Y 580.277,Z 383.202,A -85,B 0,C 180,E1 -1783.826,E2 -1783.826} C_VEL
LIN {X 0,Y 580.277,Z 383.202,A -85,B 0,C 180,E1 -1786.696,E2 -1786.696} C_VEL
LIN {X 0,Y 580.298,Z 383.2,A -85,B 0,C 180,E1 -1789.533,E2 -1789.533} C_VEL
LIN {X 0,Y 580.327,Z 383.198,A -85,B 0,C 180,E1 -1792.345,E2 -1792.345} C_VEL
LIN {X 0,Y 580.334,Z 383.2,A -85,B 0,C 180,E1 -1795.137,E2 -1795.137} C_VEL
LIN {X 0,Y 580.341,Z 383.198,A -85,B 0,C 180,E1 -1797.918,E2 -1797.918} C_VEL
LIN {X 0,Y 580.363,Z 383.193,A -85,B 0,C 180,E1 -1800.694,E2 -1800.694} C_VEL
LIN {X 0,Y 580.284,Z 383.201,A -85,B 0,C 180,E1 -1803.472,E2 -1803.472} C_VEL
LIN {X 0,Y 580.322,Z 383.202,A -85,B 0,C 180,E1 -1805.56,E2 -1805.56} C_VEL
LIN {X 0,Y 580.329,Z 383.199,A -85,B 0,C 180,E1 -1808.356,E2 -1808.356} C_VEL
LIN {X 0,Y 580.292,Z 383.202,A -85,B 0,C 180,E1 -1811.191,E2 -1811.191} C_VEL
LIN {X 0,Y 580.321,Z 383.197,A -85,B 0,C 180,E1 -1814.017,E2 -1814.017} C_VEL
LIN {X 0,Y 580.307,Z 383.199,A -85,B 0,C 180,E1 -1816.915,E2 -1816.915} C_VEL
LIN {X 0,Y 580.304,Z 383.199,A -85,B 0,C 180,E1 -1819.823,E2 -1819.823} C_VEL
LIN {X 0,Y 580.269,Z 383.208,A -85,B 0,C 180,E1 -1822.053,E2 -1822.053} C_VEL
LIN {X 0,Y 580.302,Z 383.203,A -85,B 0,C 180,E1 -1825.08,E2 -1825.08} C_VEL
LIN {X 0,Y 580.314,Z 383.202,A -85,B 0,C 180,E1 -1827.864,E2 -1827.864} C_VEL
LIN {X 0,Y 580.295,Z 383.203,A -85,B 0,C 180,E1 -1830.698,E2 -1830.698} C_VEL
LIN {X 0,Y 580.3,Z 383.199,A -85,B 0,C 180,E1 -1833.317,E2 -1833.317} C_VEL
LIN {X 0,Y 580.324,Z 383.197,A -85,B 0,C 180,E1 -1835.768,E2 -1835.768} C_VEL
LIN {X 0,Y 580.287,Z 383.203,A -85,B 0,C 180,E1 -1838.147,E2 -1838.147} C_VEL
LIN {X 0,Y 580.298,Z 383.2,A -85,B 0,C 180,E1 -1840.844,E2 -1840.844} C_VEL
LIN {X 0,Y 580.285,Z 383.201,A -85,B 0,C 180,E1 -1843.658,E2 -1843.658} C_VEL
LIN {X 0,Y 580.284,Z 383.201,A -85,B 0,C 180,E1 -1846.609,E2 -1846.609} C_VEL
LIN {X 0,Y 580.301,Z 383.202,A -85,B 0,C 180,E1 -1849.158,E2 -1849.158} C_VEL
LIN {X 0,Y 580.291,Z 383.206,A -85,B 0,C 180,E1 -1851.927,E2 -1851.927} C_VEL
LIN {X 0,Y 580.309,Z 383.315,A -85,B 0,C 180,E1 -1853.853,E2 -1853.853} C_VEL
LIN {X 0,Y 580.555,Z 387.299,A -85,B 0,C 180,E1 -1855.405,E2 -1855.405} C_VEL
LIN {X 0,Y 580.478,Z 394.032,A -85,B 0,C 180,E1 -1857.942,E2 -1857.942} C_VEL
LIN {X 0,Y 580.429,Z 401.6,A -85,B 0,C 180,E1 -1860.669,E2 -1860.669} C_VEL
LIN {X 0,Y 580.355,Z 410.215,A -85,B 0,C 180,E1 -1863.654,E2 -1863.654} C_VEL
LIN {X 0,Y 580.301,Z 418.336,A -85,B 0,C 180,E1 -1866.443,E2 -1866.443} C_VEL
LIN {X 0,Y 580.245,Z 427.24,A -85,B 0,C 180,E1 -1869.436,E2 -1869.436} C_VEL
LIN {X 0,Y 580.205,Z 436.144,A -85,B 0,C 180,E1 -1872.373,E2 -1872.373} C_VEL
LIN {X 0,Y 580.147,Z 445.049,A -85,B 0,C 180,E1 -1875.262,E2 -1875.262} C_VEL
LIN {X 0,Y 580.131,Z 452.492,A -85,B 0,C 180,E1 -1877.649,E2 -1877.649} C_VEL
LIN {X 0,Y 580.808,Z 457.236,A -85,B 0,C 180,E1 -1877.753,E2 -1877.753} C_VEL
LIN {X 0,Y 580.729,Z 470.502,A -85,B 0,C 180,E1 -1878.083,E2 -1878.083} C_VEL
LIN {X 0,Y 580.628,Z 482.321,A -85,B 0,C 180,E1 -1878.515,E2 -1878.515} C_VEL
LIN {X 0,Y 580.561,Z 494.213,A -85,B 0,C 180,E1 -1879.097,E2 -1879.097} C_VEL
LIN {X 0,Y 580.452,Z 505.481,A -85,B 0,C 180,E1 -1879.801,E2 -1879.801} C_VEL
LIN {X 0,Y 580.352,Z 515.648,A -85,B 0,C 180,E1 -1880.591,E2 -1880.591} C_VEL
LIN {X 0,Y 580.279,Z 524.787,A -85,B 0,C 180,E1 -1881.468,E2 -1881.468} C_VEL
LIN {X 0,Y 580.199,Z 533.69,A -85,B 0,C 180,E1 -1882.518,E2 -1882.518} C_VEL
LIN {X 0,Y 580.12,Z 540.465,A -85,B 0,C 180,E1 -1883.505,E2 -1883.505} C_VEL
LIN {X 0,Y 580.139,Z 545.68,A -85,B 0,C 180,E1 -1884.438,E2 -1884.438} C_VEL
LIN {X 0,Y 580.108,Z 550.371,A -85,B 0,C 180,E1 -1885.483,E2 -1885.483} C_VEL
LIN {X 0,Y 580.123,Z 553.957,A -85,B 0,C 180,E1 -1886.527,E2 -1886.527} C_VEL
LIN {X 0,Y 580.043,Z 555.808,A -85,B 0,C 180,E1 -1887.222,E2 -1887.222} C_VEL
LIN {X 0,Y 580.04,Z 557.199,A -85,B 0,C 180,E1 -1887.917,E2 -1887.917} C_VEL
LIN {X 0,Y 580.04,Z 558.784,A -85,B 0,C 180,E1 -1889.306,E2 -1889.306} C_VEL
LIN {X 0,Y 580.037,Z 559,A -85,B 0,C 180,E1 -1890,E2 -1890} C_VEL
LIN {X 0,Y 580.047,Z 558.186,A -85,B 0,C 180,E1 -1891.388,E2 -1891.388} C_VEL
LIN {X 0,Y 580.04,Z 557.201,A -85,B 0,C 180,E1 -1892.083,E2 -1892.083} C_VEL
LIN {X 0,Y 580.043,Z 555.81,A -85,B 0,C 180,E1 -1892.778,E2 -1892.778} C_VEL
LIN {X 0,Y 580.109,Z 552.897,A -85,B 0,C 180,E1 -1893.82,E2 -1893.82} C_VEL
LIN {X 0,Y 580.054,Z 548.95,A -85,B 0,C 180,E1 -1894.865,E2 -1894.865} C_VEL
LIN {X 0,Y 580.139,Z 542.879,A -85,B 0,C 180,E1 -1896.085,E2 -1896.085} C_VEL
LIN {X 0,Y 580.184,Z 536.239,A -85,B 0,C 180,E1 -1897.132,E2 -1897.132} C_VEL
LIN {X 0,Y 580.25,Z 527.993,A -85,B 0,C 180,E1 -1898.182,E2 -1898.182} C_VEL
LIN {X 0,Y 580.308,Z 519.541,A -85,B 0,C 180,E1 -1899.058,E2 -1899.058} C_VEL
LIN {X 0,Y 580.425,Z 509.1,A -85,B 0,C 180,E1 -1899.935,E2 -1899.935} C_VEL
LIN {X 0,Y 580.491,Z 498.763,A -85,B 0,C 180,E1 -1900.639,E2 -1900.639} C_VEL
LIN {X 0,Y 580.596,Z 487.253,A -85,B 0,C 180,E1 -1901.264,E2 -1901.264} C_VEL
LIN {X 0,Y 580.67,Z 474.482,A -85,B 0,C 180,E1 -1901.785,E2 -1901.785} C_VEL
LIN {X 0,Y 580.77,Z 461.451,A -85,B 0,C 180,E1 -1902.159,E2 -1902.159} C_VEL
LIN {X 0,Y 580.633,Z 455.678,A -85,B 0,C 180,E1 -1902.281,E2 -1902.281} C_VEL
LIN {X 0,Y 580.131,Z 452.493,A -85,B 0,C 180,E1 -1902.35,E2 -1902.35} C_VEL
LIN {X 0,Y 580.158,Z 443.936,A -85,B 0,C 180,E1 -1905.096,E2 -1905.096} C_VEL
LIN {X 0,Y 580.208,Z 435.032,A -85,B 0,C 180,E1 -1907.991,E2 -1907.991} C_VEL
LIN {X 0,Y 580.244,Z 427.241,A -85,B 0,C 180,E1 -1910.563,E2 -1910.563} C_VEL
LIN {X 0,Y 580.3,Z 418.337,A -85,B 0,C 180,E1 -1913.556,E2 -1913.556} C_VEL
LIN {X 0,Y 580.354,Z 410.211,A -85,B 0,C 180,E1 -1916.346,E2 -1916.346} C_VEL
LIN {X 0,Y 580.459,Z 401.585,A -85,B 0,C 180,E1 -1919.337,E2 -1919.337} C_VEL
LIN {X 0,Y 580.481,Z 393.693,A -85,B 0,C 180,E1 -1922.188,E2 -1922.188} C_VEL
LIN {X 0,Y 580.558,Z 387.071,A -85,B 0,C 180,E1 -1924.677,E2 -1924.677} C_VEL
LIN {X 0,Y 580.317,Z 383.201,A -85,B 0,C 180,E1 -1926.23,E2 -1926.23} C_VEL
LIN {X 0,Y 580.307,Z 383.202,A -85,B 0,C 180,E1 -1929.186,E2 -1929.186} C_VEL
LIN {X 0,Y 580.311,Z 383.194,A -85,B 0,C 180,E1 -1931.765,E2 -1931.765} C_VEL
LIN {X 0,Y 580.265,Z 383.206,A -85,B 0,C 180,E1 -1934.625,E2 -1934.625} C_VEL
LIN {X 0,Y 580.277,Z 383.2,A -85,B 0,C 180,E1 -1937.293,E2 -1937.293} C_VEL
LIN {X 0,Y 580.291,Z 383.198,A -85,B 0,C 180,E1 -1940.067,E2 -1940.067} C_VEL
LIN {X 0,Y 580.297,Z 383.198,A -85,B 0,C 180,E1 -1943.064,E2 -1943.064} C_VEL
LIN {X 0,Y 580.3,Z 383.195,A -85,B 0,C 180,E1 -1945.439,E2 -1945.439} C_VEL
LIN {X 0,Y 580.302,Z 383.199,A -85,B 0,C 180,E1 -1947.967,E2 -1947.967} C_VEL
LIN {X 0,Y 580.3,Z 383.199,A -85,B 0,C 180,E1 -1950.688,E2 -1950.688} C_VEL
LIN {X 0,Y 580.275,Z 383.199,A -85,B 0,C 180,E1 -1953.376,E2 -1953.376} C_VEL
LIN {X 0,Y 580.295,Z 383.199,A -85,B 0,C 180,E1 -1955.683,E2 -1955.683} C_VEL
LIN {X 0,Y 580.267,Z 383.208,A -85,B 0,C 180,E1 -1957.947,E2 -1957.947} C_VEL
LIN {X 0,Y 580.309,Z 383.194,A -85,B 0,C 180,E1 -1960.914,E2 -1960.914} C_VEL
LIN {X 0,Y 580.276,Z 383.207,A -85,B 0,C 180,E1 -1963.825,E2 -1963.825} C_VEL
LIN {X 0,Y 580.274,Z 383.199,A -85,B 0,C 180,E1 -1966.696,E2 -1966.696} C_VEL
LIN {X 0,Y 580.295,Z 383.205,A -85,B 0,C 180,E1 -1969.533,E2 -1969.533} C_VEL
LIN {X 0,Y 580.324,Z 383.193,A -85,B 0,C 180,E1 -1972.344,E2 -1972.344} C_VEL
LIN {X 0,Y 580.338,Z 383.196,A -85,B 0,C 180,E1 -1975.137,E2 -1975.137} C_VEL
LIN {X 0,Y 580.33,Z 383.194,A -85,B 0,C 180,E1 -1977.918,E2 -1977.918} C_VEL
LIN {X 0,Y 580.359,Z 383.19,A -85,B 0,C 180,E1 -1980.694,E2 -1980.694} C_VEL
LIN {X 0,Y 580.29,Z 383.201,A -85,B 0,C 180,E1 -1983.472,E2 -1983.472} C_VEL
LIN {X 0,Y 580.323,Z 383.195,A -85,B 0,C 180,E1 -1985.56,E2 -1985.56} C_VEL
LIN {X 0,Y 580.327,Z 383.194,A -85,B 0,C 180,E1 -1988.356,E2 -1988.356} C_VEL
LIN {X 0,Y 580.323,Z 383.197,A -85,B 0,C 180,E1 -1991.208,E2 -1991.208} C_VEL
LIN {X 0,Y 580.306,Z 383.198,A -85,B 0,C 180,E1 -1994.339,E2 -1994.339} C_VEL
LIN {X 0,Y 580.309,Z 383.2,A -85,B 0,C 180,E1 -1996.916,E2 -1996.916} C_VEL
LIN {X 0,Y 580.302,Z 383.196,A -85,B 0,C 180,E1 -1999.822,E2 -1999.822} C_VEL
LIN {X 0,Y 580.282,Z 383.198,A -85,B 0,C 180,E1 -2001.341,E2 -2001.341} C_VEL
LIN {X 0,Y 579.592,Z 383.286,A -85,B 0,C 180,E1 -2001.92,E2 -2001.92} C_VEL
LIN {X 0,Y 576.72,Z 383.645,A -85,B 0,C 180,E1 -2002.86,E2 -2002.86} C_VEL
LIN {X 0,Y 574.322,Z 383.942,A -85,B 0,C 180,E1 -2003.617,E2 -2003.617} C_VEL
LIN {X 0,Y 573.317,Z 384.072,A -85,B 0,C 180,E1 -2004.201,E2 -2004.201} C_VEL
LIN {X 0,Y 573.247,Z 384.077,A -85,B 0,C 180,E1 -2004.399,E2 -2004.399} C_VEL
LIN {X 0,Y 573.26,Z 384.074,A -85,B 0,C 180,E1 -2006.975,E2 -2006.975} C_VEL
LIN {X 0,Y 573.247,Z 384.075,A -85,B 0,C 180,E1 -2009.49,E2 -2009.49} C_VEL
LIN {X 0,Y 573.249,Z 384.082,A -85,B 0,C 180,E1 -2012.23,E2 -2012.23} C_VEL
LIN {X 0,Y 573.246,Z 384.075,A -85,B 0,C 180,E1 -2014.775,E2 -2014.775} C_VEL
LIN {X 0,Y 573.248,Z 384.074,A -85,B 0,C 180,E1 -2017.167,E2 -2017.167} C_VEL
LIN {X 0,Y 573.243,Z 384.079,A -85,B 0,C 180,E1 -2019.607,E2 -2019.607} C_VEL
LIN {X 0,Y 573.237,Z 384.075,A -85,B 0,C 180,E1 -2022.643,E2 -2022.643} C_VEL
LIN {X 0,Y 573.234,Z 384.085,A -85,B 0,C 180,E1 -2025.668,E2 -2025.668} C_VEL
LIN {X 0,Y 573.241,Z 384.074,A -85,B 0,C 180,E1 -2028.545,E2 -2028.545} C_VEL
LIN {X 0,Y 573.245,Z 384.081,A -85,B 0,C 180,E1 -2031.3,E2 -2031.3} C_VEL
LIN {X 0,Y 573.261,Z 384.073,A -85,B 0,C 180,E1 -2034.012,E2 -2034.012} C_VEL
LIN {X 0,Y 573.282,Z 384.07,A -85,B 0,C 180,E1 -2036.52,E2 -2036.52} C_VEL
LIN {X 0,Y 573.237,Z 384.083,A -85,B 0,C 180,E1 -2039.116,E2 -2039.116} C_VEL
LIN {X 0,Y 573.263,Z 384.072,A -85,B 0,C 180,E1 -2041.969,E2 -2041.969} C_VEL
LIN {X 0,Y 573.256,Z 384.076,A -85,B 0,C 180,E1 -2044.591,E2 -2044.591} C_VEL
LIN {X 0,Y 573.235,Z 384.076,A -85,B 0,C 180,E1 -2047.663,E2 -2047.663} C_VEL
LIN {X 0,Y 573.206,Z 384.086,A -85,B 0,C 180,E1 -2048.721,E2 -2048.721} C_VEL
LIN {X 0,Y 573.177,Z 388.312,A -85,B 0,C 180,E1 -2051.41,E2 -2051.41} C_VEL
LIN {X 0,Y 573.145,Z 392.028,A -85,B 0,C 180,E1 -2053.619,E2 -2053.619} C_VEL
LIN {X 0,Y 573.116,Z 396.978,A -85,B 0,C 180,E1 -2056.527,E2 -2056.527} C_VEL
LIN {X 0,Y 573.087,Z 401.902,A -85,B 0,C 180,E1 -2059.4,E2 -2059.4} C_VEL
LIN {X 0,Y 573.082,Z 407.033,A -85,B 0,C 180,E1 -2062.248,E2 -2062.248} C_VEL
LIN {X 0,Y 573.07,Z 412.25,A -85,B 0,C 180,E1 -2065.076,E2 -2065.076} C_VEL
LIN {X 0,Y 572.989,Z 417.537,A -85,B 0,C 180,E1 -2067.891,E2 -2067.891} C_VEL
LIN {X 0,Y 572.981,Z 422.886,A -85,B 0,C 180,E1 -2070.703,E2 -2070.703} C_VEL
LIN {X 0,Y 573.004,Z 424.528,A -85,B 0,C 180,E1 -2071.56,E2 -2071.56} C_VEL
LIN {X 0,Y 573.848,Z 431.282,A -85,B 0,C 180,E1 -2071.733,E2 -2071.733} C_VEL
LIN {X 0,Y 573.717,Z 444.216,A -85,B 0,C 180,E1 -2072.106,E2 -2072.106} C_VEL
LIN {X 0,Y 573.621,Z 457.064,A -85,B 0,C 180,E1 -2072.633,E2 -2072.633} C_VEL
LIN {X 0,Y 573.523,Z 468.349,A -85,B 0,C 180,E1 -2073.249,E2 -2073.249} C_VEL
LIN {X 0,Y 573.368,Z 479.826,A -85,B 0,C 180,E1 -2074.042,E2 -2074.042} C_VEL
LIN {X 0,Y 573.252,Z 490.045,A -85,B 0,C 180,E1 -2074.923,E2 -2074.923} C_VEL
LIN {X 0,Y 573.158,Z 499.846,A -85,B 0,C 180,E1 -2075.983,E2 -2075.983} C_VEL
LIN {X 0,Y 573.133,Z 507.757,A -85,B 0,C 180,E1 -2077.044,E2 -2077.044} C_VEL
LIN {X 0,Y 573.05,Z 514.107,A -85,B 0,C 180,E1 -2078.108,E2 -2078.108} C_VEL
LIN {X 0,Y 572.991,Z 519.173,A -85,B 0,C 180,E1 -2079.175,E2 -2079.175} C_VEL
LIN {X 0,Y 572.991,Z 523.101,A -85,B 0,C 180,E1 -2080.244,E2 -2080.244} C_VEL
LIN {X 0,Y 572.975,Z 525.994,A -85,B 0,C 180,E1 -2081.318,E2 -2081.318} C_VEL
LIN {X 0,Y 572.946,Z 527.359,A -85,B 0,C 180,E1 -2082.036,E2 -2082.036} C_VEL
LIN {X 0,Y 572.945,Z 528.315,A -85,B 0,C 180,E1 -2082.756,E2 -2082.756} C_VEL
LIN {X 0,Y 572.968,Z 528.87,A -85,B 0,C 180,E1 -2083.477,E2 -2083.477} C_VEL
LIN {X 0,Y 572.961,Z 528.95,A -85,B 0,C 180,E1 -2084.299,E2 -2084.299} C_VEL
LIN {X 0,Y 572.916,Z 527.952,A -85,B 0,C 180,E1 -2085.657,E2 -2085.657} C_VEL
LIN {X 0,Y 572.941,Z 525.692,A -85,B 0,C 180,E1 -2086.905,E2 -2086.905} C_VEL
LIN {X 0,Y 572.997,Z 521.816,A -85,B 0,C 180,E1 -2088.226,E2 -2088.226} C_VEL
LIN {X 0,Y 573.041,Z 517.297,A -85,B 0,C 180,E1 -2089.338,E2 -2089.338} C_VEL
LIN {X 0,Y 573.067,Z 511.435,A -85,B 0,C 180,E1 -2090.458,E2 -2090.458} C_VEL
LIN {X 0,Y 573.124,Z 503.96,A -85,B 0,C 180,E1 -2091.585,E2 -2091.585} C_VEL
LIN {X 0,Y 573.204,Z 496.202,A -85,B 0,C 180,E1 -2092.529,E2 -2092.529} C_VEL
LIN {X 0,Y 573.307,Z 487.085,A -85,B 0,C 180,E1 -2093.44,E2 -2093.44} C_VEL
LIN {X 0,Y 573.361,Z 477.265,A -85,B 0,C 180,E1 -2094.244,E2 -2094.244} C_VEL
LIN {X 0,Y 573.52,Z 466.863,A -85,B 0,C 180,E1 -2094.932,E2 -2094.932} C_VEL
LIN {X 0,Y 573.607,Z 454.208,A -85,B 0,C 180,E1 -2095.587,E2 -2095.587} C_VEL
LIN {X 0,Y 573.757,Z 441.773,A -85,B 0,C 180,E1 -2096.067,E2 -2096.067} C_VEL
LIN {X 0,Y 573.769,Z 429.397,A -85,B 0,C 180,E1 -2096.402,E2 -2096.402} C_VEL
LIN {X 0,Y 572.994,Z 424.522,A -85,B 0,C 180,E1 -2096.534,E2 -2096.534} C_VEL
LIN {X 0,Y 572.978,Z 418.973,A -85,B 0,C 180,E1 -2099.44,E2 -2099.44} C_VEL
LIN {X 0,Y 573.042,Z 412.915,A -85,B 0,C 180,E1 -2102.658,E2 -2102.658} C_VEL
LIN {X 0,Y 573.066,Z 406.634,A -85,B 0,C 180,E1 -2106.062,E2 -2106.062} C_VEL
LIN {X 0,Y 573.053,Z 401.874,A -85,B 0,C 180,E1 -2108.716,E2 -2108.716} C_VEL
LIN {X 0,Y 573.096,Z 396.993,A -85,B 0,C 180,E1 -2111.578,E2 -2111.578} C_VEL
LIN {X 0,Y 573.2,Z 391.716,A -85,B 0,C 180,E1 -2114.673,E2 -2114.673} C_VEL
LIN {X 0,Y 573.19,Z 386.835,A -85,B 0,C 180,E1 -2117.595,E2 -2117.595} C_VEL
LIN {X 0,Y 573.193,Z 384.088,A -85,B 0,C 180,E1 -2119.48,E2 -2119.48} C_VEL
LIN {X 0,Y 573.233,Z 384.086,A -85,B 0,C 180,E1 -2122.192,E2 -2122.192} C_VEL
LIN {X 0,Y 573.265,Z 384.078,A -85,B 0,C 180,E1 -2124.816,E2 -2124.816} C_VEL
LIN {X 0,Y 573.25,Z 384.078,A -85,B 0,C 180,E1 -2127.355,E2 -2127.355} C_VEL
LIN {X 0,Y 573.251,Z 384.081,A -85,B 0,C 180,E1 -2129.824,E2 -2129.824} C_VEL
LIN {X 0,Y 573.284,Z 384.074,A -85,B 0,C 180,E1 -2132.235,E2 -2132.235} C_VEL
LIN {X 0,Y 573.264,Z 384.076,A -85,B 0,C 180,E1 -2135.121,E2 -2135.121} C_VEL
LIN {X 0,Y 573.232,Z 384.08,A -85,B 0,C 180,E1 -2137.662,E2 -2137.662} C_VEL
LIN {X 0,Y 573.271,Z 384.075,A -85,B 0,C 180,E1 -2140.728,E2 -2140.728} C_VEL
LIN {X 0,Y 573.253,Z 384.077,A -85,B 0,C 180,E1 -2143.622,E2 -2143.622} C_VEL
LIN {X 0,Y 573.234,Z 384.08,A -85,B 0,C 180,E1 -2146.53,E2 -2146.53} C_VEL
LIN {X 0,Y 573.276,Z 384.075,A -85,B 0,C 180,E1 -2148.734,E2 -2148.734} C_VEL
LIN {X 0,Y 573.301,Z 384.071,A -85,B 0,C 180,E1 -2151.541,E2 -2151.541} C_VEL
LIN {X 0,Y 573.29,Z 384.072,A -85,B 0,C 180,E1 -2154.372,E2 -2154.372} C_VEL
LIN {X 0,Y 573.311,Z 384.073,A -85,B 0,C 180,E1 -2157.893,E2 -2157.893} C_VEL
LIN {X 0,Y 573.333,Z 384.069,A -85,B 0,C 180,E1 -2160.702,E2 -2160.702} C_VEL
LIN {X 0,Y 573.236,Z 384.079,A -85,B 0,C 180,E1 -2163.515,E2 -2163.515} C_VEL
LIN {X 0,Y 573.288,Z 384.077,A -85,B 0,C 180,E1 -2165.628,E2 -2165.628} C_VEL
LIN {X 0,Y 573.301,Z 384.075,A -85,B 0,C 180,E1 -2168.459,E2 -2168.459} C_VEL
LIN {X 0,Y 573.264,Z 384.079,A -85,B 0,C 180,E1 -2171.312,E2 -2171.312} C_VEL
LIN {X 0,Y 573.267,Z 384.077,A -85,B 0,C 180,E1 -2174.193,E2 -2174.193} C_VEL
LIN {X 0,Y 573.254,Z 384.079,A -85,B 0,C 180,E1 -2177.112,E2 -2177.112} C_VEL
LIN {X 0,Y 573.253,Z 384.079,A -85,B 0,C 180,E1 -2180.077,E2 -2180.077} C_VEL
LIN {X 0,Y 573.232,Z 384.081,A -85,B 0,C 180,E1 -2182.338,E2 -2182.338} C_VEL
LIN {X 0,Y 573.25,Z 384.078,A -85,B 0,C 180,E1 -2185.41,E2 -2185.41} C_VEL
LIN {X 0,Y 573.259,Z 384.081,A -85,B 0,C 180,E1 -2188.032,E2 -2188.032} C_VEL
LIN {X 0,Y 573.241,Z 384.084,A -85,B 0,C 180,E1 -2190.886,E2 -2190.886} C_VEL
LIN {X 0,Y 573.257,Z 384.078,A -85,B 0,C 180,E1 -2193.525,E2 -2193.525} C_VEL
LIN {X 0,Y 573.258,Z 384.076,A -85,B 0,C 180,E1 -2196.049,E2 -2196.049} C_VEL
LIN {X 0,Y 573.247,Z 384.079,A -85,B 0,C 180,E1 -2198.701,E2 -2198.701} C_VEL
LIN {X 0,Y 573.252,Z 384.081,A -85,B 0,C 180,E1 -2201.596,E2 -2201.596} C_VEL
LIN {X 0,Y 573.237,Z 384.084,A -85,B 0,C 180,E1 -2204.334,E2 -2204.334} C_VEL
LIN {X 0,Y 573.243,Z 384.084,A -85,B 0,C 180,E1 -2207.359,E2 -2207.359} C_VEL
LIN {X 0,Y 573.248,Z 384.082,A -85,B 0,C 180,E1 -2210.394,E2 -2210.394} C_VEL
LIN {X 0,Y 573.26,Z 384.082,A -85,B 0,C 180,E1 -2213.517,E2 -2213.517} C_VEL
LIN {X 0,Y 573.293,Z 384.315,A -85,B 0,C 180,E1 -2213.737,E2 -2213.737} C_VEL
LIN {X 0,Y 573.549,Z 387.9,A -85,B 0,C 180,E1 -2215.184,E2 -2215.184} C_VEL
LIN {X 0,Y 573.476,Z 394.65,A -85,B 0,C 180,E1 -2217.737,E2 -2217.737} C_VEL
LIN {X 0,Y 573.403,Z 402.522,A -85,B 0,C 180,E1 -2220.642,E2 -2220.642} C_VEL
LIN {X 0,Y 573.317,Z 410.679,A -85,B 0,C 180,E1 -2223.492,E2 -2223.492} C_VEL
LIN {X 0,Y 573.266,Z 418.336,A -85,B 0,C 180,E1 -2226.136,E2 -2226.136} C_VEL
LIN {X 0,Y 573.229,Z 425.888,A -85,B 0,C 180,E1 -2228.716,E2 -2228.716} C_VEL
LIN {X 0,Y 573.158,Z 433.918,A -85,B 0,C 180,E1 -2231.409,E2 -2231.409} C_VEL
LIN {X 0,Y 573.11,Z 442.823,A -85,B 0,C 180,E1 -2234.349,E2 -2234.349} C_VEL
LIN {X 0,Y 573.081,Z 452.283,A -85,B 0,C 180,E1 -2237.427,E2 -2237.427} C_VEL
LIN {X 0,Y 573.089,Z 452.492,A -85,B 0,C 180,E1 -2237.495,E2 -2237.495} C_VEL
LIN {X 0,Y 573.878,Z 459.516,A -85,B 0,C 180,E1 -2237.647,E2 -2237.647} C_VEL
LIN {X 0,Y 573.762,Z 471.88,A -85,B 0,C 180,E1 -2237.981,E2 -2237.981} C_VEL
LIN {X 0,Y 573.67,Z 484.286,A -85,B 0,C 180,E1 -2238.462,E2 -2238.462} C_VEL
LIN {X 0,Y 573.585,Z 495.783,A -85,B 0,C 180,E1 -2239.052,E2 -2239.052} C_VEL
LIN {X 0,Y 573.445,Z 506.748,A -85,B 0,C 180,E1 -2239.764,E2 -2239.764} C_VEL
LIN {X 0,Y 573.308,Z 515.648,A -85,B 0,C 180,E1 -2240.474,E2 -2240.474} C_VEL
LIN {X 0,Y 573.215,Z 524.787,A -85,B 0,C 180,E1 -2241.362,E2 -2241.362} C_VEL
LIN {X 0,Y 573.142,Z 533.69,A -85,B 0,C 180,E1 -2242.425,E2 -2242.425} C_VEL
LIN {X 0,Y 573.051,Z 540.405,A -85,B 0,C 180,E1 -2243.415,E2 -2243.415} C_VEL
LIN {X 0,Y 573.07,Z 545.68,A -85,B 0,C 180,E1 -2244.37,E2 -2244.37} C_VEL
LIN {X 0,Y 573.028,Z 550.372,A -85,B 0,C 180,E1 -2245.427,E2 -2245.427} C_VEL
LIN {X 0,Y 573.022,Z 553.957,A -85,B 0,C 180,E1 -2246.484,E2 -2246.484} C_VEL
LIN {X 0,Y 572.959,Z 555.808,A -85,B 0,C 180,E1 -2247.188,E2 -2247.188} C_VEL
LIN {X 0,Y 572.939,Z 557.199,A -85,B 0,C 180,E1 -2247.891,E2 -2247.891} C_VEL
LIN {X 0,Y 572.941,Z 558.785,A -85,B 0,C 180,E1 -2249.297,E2 -2249.297} C_VEL
LIN {X 0,Y 572.938,Z 559,A -85,B 0,C 180,E1 -2250,E2 -2250} C_VEL
LIN {X 0,Y 572.946,Z 558.186,A -85,B 0,C 180,E1 -2251.406,E2 -2251.406} C_VEL
LIN {X 0,Y 572.939,Z 557.2,A -85,B 0,C 180,E1 -2252.109,E2 -2252.109} C_VEL
LIN {X 0,Y 572.959,Z 555.81,A -85,B 0,C 180,E1 -2252.812,E2 -2252.812} C_VEL
LIN {X 0,Y 573.014,Z 552.896,A -85,B 0,C 180,E1 -2253.868,E2 -2253.868} C_VEL
LIN {X 0,Y 572.963,Z 548.95,A -85,B 0,C 180,E1 -2254.925,E2 -2254.925} C_VEL
LIN {X 0,Y 573.064,Z 542.878,A -85,B 0,C 180,E1 -2256.16,E2 -2256.16} C_VEL
LIN {X 0,Y 573.119,Z 536.239,A -85,B 0,C 180,E1 -2257.22,E2 -2257.22} C_VEL
LIN {X 0,Y 573.201,Z 527.993,A -85,B 0,C 180,E1 -2258.283,E2 -2258.283} C_VEL
LIN {X 0,Y 573.287,Z 519.542,A -85,B 0,C 180,E1 -2259.17,E2 -2259.17} C_VEL
LIN {X 0,Y 573.429,Z 509.102,A -85,B 0,C 180,E1 -2260.058,E2 -2260.058} C_VEL
LIN {X 0,Y 573.546,Z 497.439,A -85,B 0,C 180,E1 -2260.852,E2 -2260.852} C_VEL
LIN {X 0,Y 573.651,Z 486.309,A -85,B 0,C 180,E1 -2261.446,E2 -2261.446} C_VEL
LIN {X 0,Y 573.753,Z 473.184,A -85,B 0,C 180,E1 -2261.974,E2 -2261.974} C_VEL
LIN {X 0,Y 573.868,Z 460.536,A -85,B 0,C 180,E1 -2262.33,E2 -2262.33} C_VEL
LIN {X 0,Y 573.486,Z 455.251,A -85,B 0,C 180,E1 -2262.445,E2 -2262.445} C_VEL
LIN {X 0,Y 573.089,Z 452.493,A -85,B 0,C 180,E1 -2262.505,E2 -2262.505} C_VEL
LIN {X 0,Y 573.087,Z 443.936,A -85,B 0,C 180,E1 -2265.287,E2 -2265.287} C_VEL
LIN {X 0,Y 573.147,Z 436.145,A -85,B 0,C 180,E1 -2267.851,E2 -2267.851} C_VEL
LIN {X 0,Y 573.2,Z 428.354,A -85,B 0,C 180,E1 -2270.452,E2 -2270.452} C_VEL
LIN {X 0,Y 573.222,Z 420.442,A -85,B 0,C 180,E1 -2273.141,E2 -2273.141} C_VEL
LIN {X 0,Y 573.291,Z 412.731,A -85,B 0,C 180,E1 -2275.797,E2 -2275.797} C_VEL
LIN {X 0,Y 573.367,Z 404.828,A -85,B 0,C 180,E1 -2278.557,E2 -2278.557} C_VEL
LIN {X 0,Y 573.408,Z 398.099,A -85,B 0,C 180,E1 -2280.982,E2 -2280.982} C_VEL
LIN {X 0,Y 573.545,Z 391.175,A -85,B 0,C 180,E1 -2283.566,E2 -2283.566} C_VEL
LIN {X 0,Y 573.55,Z 385.982,A -85,B 0,C 180,E1 -2285.581,E2 -2285.581} C_VEL
LIN {X 0,Y 573.304,Z 384.075,A -85,B 0,C 180,E1 -2286.37,E2 -2286.37} C_VEL
LIN {X 0,Y 573.246,Z 384.076,A -85,B 0,C 180,E1 -2289.606,E2 -2289.606} C_VEL
LIN {X 0,Y 573.248,Z 384.08,A -85,B 0,C 180,E1 -2292.642,E2 -2292.642} C_VEL
LIN {X 0,Y 573.235,Z 384.076,A -85,B 0,C 180,E1 -2295.666,E2 -2295.666} C_VEL
LIN {X 0,Y 573.242,Z 384.082,A -85,B 0,C 180,E1 -2298.544,E2 -2298.544} C_VEL
LIN {X 0,Y 573.245,Z 384.075,A -85,B 0,C 180,E1 -2301.298,E2 -2301.298} C_VEL
LIN {X 0,Y 573.26,Z 384.075,A -85,B 0,C 180,E1 -2304.01,E2 -2304.01} C_VEL
LIN {X 0,Y 573.278,Z 384.078,A -85,B 0,C 180,E1 -2306.518,E2 -2306.518} C_VEL
LIN {X 0,Y 573.238,Z 384.076,A -85,B 0,C 180,E1 -2309.114,E2 -2309.114} C_VEL
LIN {X 0,Y 573.257,Z 384.078,A -85,B 0,C 180,E1 -2311.968,E2 -2311.968} C_VEL
LIN {X 0,Y 573.248,Z 384.077,A -85,B 0,C 180,E1 -2314.589,E2 -2314.589} C_VEL
LIN {X 0,Y 573.23,Z 384.08,A -85,B 0,C 180,E1 -2317.662,E2 -2317.662} C_VEL
LIN {X 0,Y 573.269,Z 384.072,A -85,B 0,C 180,E1 -2320.728,E2 -2320.728} C_VEL
LIN {X 0,Y 573.251,Z 384.08,A -85,B 0,C 180,E1 -2323.622,E2 -2323.622} C_VEL
LIN {X 0,Y 573.231,Z 384.077,A -85,B 0,C 180,E1 -2326.529,E2 -2326.529} C_VEL
LIN {X 0,Y 573.252,Z 384.074,A -85,B 0,C 180,E1 -2328.745,E2 -2328.745} C_VEL
LIN {X 0,Y 573.298,Z 384.076,A -85,B 0,C 180,E1 -2331.541,E2 -2331.541} C_VEL
LIN {X 0,Y 573.286,Z 384.069,A -85,B 0,C 180,E1 -2334.372,E2 -2334.372} C_VEL
LIN {X 0,Y 573.301,Z 384.069,A -85,B 0,C 180,E1 -2337.892,E2 -2337.892} C_VEL
LIN {X 0,Y 573.329,Z 384.066,A -85,B 0,C 180,E1 -2340.702,E2 -2340.702} C_VEL
LIN {X 0,Y 573.241,Z 384.079,A -85,B 0,C 180,E1 -2343.514,E2 -2343.514} C_VEL
